// ---- Data types/METS/_StationOperational/C715 Tempalate Example/E_04_ElevatorState_C715.TcDUT
TYPE E_04_ElevatorState_C715 :
(
	SEQ_04_INIT									:=0,
	SEQ_04_ENABLEDEVICES							:=1,
	SEQ_04_HOMING								:=10,
	SEQ_04_MOVETODOWNLIMIT_DONE				:=20,
	SEQ_04_HOMINGWITHDATUM						:=30,

	SEQ_04_MOVETOHOMEPOS_TRY					:=40,
	SEQ_04_MOVETOHOMEPOS_DONE					:=50,
	SEQ_04_HOMED								:=90,
	SEQ_04_READY									:=100,

	SEQ_04_REQACCEPTED							:=110,

	SEQ_04_MOVEUP_TRY							:=120,
	SEQ_04_MOVEUP_DONE							:=130,
	SEQ_04_UNLOADBUNDLE_TRY						:=140,
	SEQ_04_UNLOADBUNDLE_DONE					:=150,

	SEQ_04_MOVEPOSITIVE_TRY						:=160,
	SEQ_04_MOVEPOSITIVE_DONE						:=170,
	SEQ_04_MOVENEGATIVE_TRY						:=180,
	SEQ_04_MOVENEGATIVE_DONE					:=190,
	SEQ_04_REJECTEXTEND_TRY						:=200,
	SEQ_04_REJECTEXTEND_DONE						:=210,
	SEQ_04_REJECTRETRACT_TRY						:=220,
	SEQ_04_REJECTRETRACT_DONE						:=230,


	(*SEQ_04_MOVEDOWN_TRY						:=160,
	SEQ_04_MOVEDOWN_DONE						:=170,*)

	SEQ_04_COMPLETE_TRY							:=340,
	SEQ_04_COMPLETE								:=350

);
END_TYPE

// ---- Data types/METS/_StationOperational/C715 Tempalate Example/E_Axis_C715.TcDUT
TYPE E_Axis_C715 :
(
	E_C715_WALKINGBEAM	:=1,
	E_C715_ELEVATOR		:=2,
	E_C715_TRANSFER		:=3,
	E_C715_PRESENTATION	:=4

);
END_TYPE

// ---- Data types/METS/_StationOperational/C715 Tempalate Example/E_Cylinder_C715.TcDUT
TYPE E_Cylinder_C715 :
(
	E_C715_STOPGATE01		:=1,
	E_C715_STOPGATE02		:=2,
	E_C715_BUNDLEALIGN	:=3,
	E_C715_TAMPHEAD		:=4,
	E_C715_LABELFORM		:=5,
	E_C715_BUNDLEREJECT	:=6,
	E_C715_BUNDLEPUSH	:=7

);
END_TYPE

// ---- Data types/METS/_StationOperational/C715 Tempalate Example/ST_04_ElevatorSeq_C715.TcDUT
  TYPE ST_04_ElevatorSeq_C715 :
STRUCT
	e04SeqState					: E_04_ElevatorState_C715;

	bSeqAbort					:BOOL;		(*Function Abort By Manager*)
	bSeqHomingRequest			:BOOL;		(*FUNCTION Homing Requested BY Manager OR Internal Functions*)
	bSeqWaitOnRequest			:BOOL;		(*Function In Valide State Avaiting For Request Command*)
	bSeqRequest					:BOOL;		(*Request Commnad To Start Function Cycle*)

	bSeqIsHoming					: BOOL;
	bSeqInProgress				:BOOL;		(*Function In Progress With Cycle*)
	bSeqComplete				:BOOL;		(*Function Complete Cycle - Flag Set After Every Cycle Finsh*)
	bSeqDone					:BOOL;		(*Function Sequence Finished With Success - Flag Set For One PLC Cycle*)
	bSeqError						: BOOL;
	nSeqErrorID					: UDINT;

	bAutoHomingAllowed			: BOOL;
	bStationHomed					:BOOL;		(*FUNCTION Homed*)
	bStationNotMoving				:BOOL;		(*Function Parts Are Not Moving*)
	bStationInPause				: BOOL;

	bMachineInError				: BOOL;
	bPassthroughMode				:BOOL;

	stBundleTracking				: ST_BundleTrackingRegister_C715;
	bTrackigDataSync				: BOOL;
	bDisableBottomLimit			: BOOL;

	bSynchroMoveActive			: BOOL;

END_STRUCT
END_TYPE

// ---- Data types/METS/_StationOperational/C715 Tempalate Example/ST_BundleTrackingRegister_C715.TcDUT
TYPE ST_BundleTrackingRegister_C715 :
STRUCT
	bOuterPresent				: BOOL;
	sOuterTimeStamp			: STRING(30);
	bOuterAligned				: BOOL;
	bLabelApplied				: BOOL;		(* TRUE = label has been printed and applied to Outer *)
	bLabelFormed				: BOOL;
	sLabelBarcode				: T_OUTER_Barcode;
	sConfirmationCode 			: T_MaxString;
	bOCVCreated				: BOOL;
	bOACCreated				: BOOL;
	bOuterIsValid				: BOOL;
	bDumpDataReq			: BOOL;
END_STRUCT
END_TYPE

// ---- Data types/METS/_StationOperational/C715 Tempalate Example/ST_CommonStationConfig_C715.TcDUT
TYPE ST_CommonStationConfig_C715 :
STRUCT

	fWalkingBeamHomeOffset		: LREAL :=55;
	fWalkingBeamVelo			: LREAL :=250;
	fWalkingBeamDistance		: LREAL :=360;

	tAlignTimeOut				: TIME  :=T#10S;

	tFormHeadTime				: TIME 	:=T#1500MS;

	fElevatorHomeOffset			: LREAL :=0;
	fElevatorMoveUpVelo			: LREAL :=400;
	fElevatorUnloadPosition		: LREAL :=310;
	fElevatorMoveDownVelo		: LREAL :=600;
	fElevatorLoadPosition		: LREAL :=0;

	tTransferTimeOut			: TIME 	:=T#10S;

	fTransferHomeOffset			: LREAL :=0;
	fTransferRejectVelo			: REAL 	:=-400;
	fTransferValidVelo			: REAL 	:=400;

	fPresentationHomeOffset		: LREAL :=0;
	fPresentationVelo			: REAL 	:=400;
	fPresentationDistance		: REAL 	:=115;

	(*bAllStationsHomed			: BOOL;
	bAllStationsCycledStopped	: BOOL;
	bCycleStopRequest			: BOOL;
	bManualModeHMI				: BOOL;
	bAllStationsOKToIndex		: BOOL;*)
END_STRUCT
END_TYPE

// ---- Data types/METS/_StationOperational/E_00_StationStateTemplate.TcDUT
TYPE E_00_StationStateTemplate :
(
	SEQ_00_INIT									:=0,
	SEQ_00_ENABLEDEVICES							:=1,
	SEQ_00_HOMING								:=10,
	SEQ_00_MOVETOHOMEPOS_TRY					:=20,
	SEQ_00_MOVETOHOMEPOS_DONE					:=30,
	SEQ_00_HOMED								:=90,
	SEQ_00_READY									:=100,

	SEQ_00_REQACCEPTED							:=110,

(***************************************************************************)
(**)
(***************************************************************************)

	SEQ_00_COMPLETE_TRY							:=340,
	SEQ_00_COMPLETE								:=350


);
END_TYPE

// ---- Data types/METS/_StationOperational/Manual Machine/E_OuterPrintStationState.TcDUT
TYPE E_OuterPrintStationState :
(
	STATION_SEQ_INIT:=100,
	STATION_SEQ_TRY_HOMING:=110,
	STATION_SEQ_HOMED:=120,
	STATION_SEQ_READY:=130,

	STATION_SEQ_GATE_DOWN_TRY:=140,
	STATION_SEQ_GATE_DOWN_DONE:=150,

	STATION_SEQ_APPLY_LABEL_TRY:=160,
	STATION_SEQ_APPLY_LABEL_DONE:=170,

	STATION_SEQ_GATE_UP_TRY:=180,
	STATION_SEQ_GATE_UP_DONE:=190,

	STATION_SEQ_COMPLETE_TRY:=200,
	STATION_SEQ_COMPLETE:=210


);
END_TYPE

// ---- Data types/METS/_StationOperational/SeqCtrl/ST_STATION_Requests.TcDUT
TYPE ST_STATION_Requests :
STRUCT

	bSeqAbort						:BOOL;		(*Function Abort By Manager*)
	bSeqInhibit						: BOOL;		(*in girafe is like bMachineInError*)
	bSeqHomingRequest			:BOOL;		(*FUNCTION Homing Requested BY Manager OR Internal Functions*)
	bSeqWaitOnRequest			:BOOL;		(*Function In Valide State Avaiting For Request Command*)
	bSeqRequest					:BOOL;		(*Request Commnad To Start Function Cycle*)

END_STRUCT
END_TYPE

// ---- Data types/METS/_StationOperational/SeqCtrl/ST_STATION_Status.TcDUT
TYPE ST_STATION_Status :
STRUCT

	bSeqIsHoming					: BOOL;
	bStationHomed					:BOOL;		(*FUNCTION Homed*)
	bSeqInProgress				:BOOL;		(*Function In Progress With Cycle*)
	bSeqComplete				:BOOL;		(*Function Complete Cycle - Flag Set After Every Cycle Finsh*)
	bSeqDone					:BOOL;		(*Function Sequence Finished With Success - Flag Set For One PLC Cycle*)
	bStationNotMoving				:BOOL;		(*Function Parts Are Not Moving*)

	bSeqError						: BOOL;
	nSeqErrorID					: UDINT;

END_STRUCT
END_TYPE

// ---- Data types/METS/_StationOperational/ST_00_StationStructTemplate.TcDUT
TYPE ST_00_StationStructTemplate :
STRUCT

	e00SeqState		: E_00_StationStateTemplate;

	REQ				: ST_STATION_Requests;
	STAT				: ST_STATION_Status;

(*Variable examles only*)
(*
	bPassthroughMode			:BOOL;

	stBundleTracking				: ST_BundleTrackingRegister;
	bTrigCamera					: BOOL;
	bCameraDone					: BOOL;


*)

END_STRUCT
END_TYPE

// ---- POUs/_Exclude/DUT/E_LOG_HandlerName_OLD.TcDUT
TYPE E_LOG_HandlerName_OLD :
(

		//E_LOG_OKCONECCTIONTOFSS,
		//E_LOG_LOSTCONECCTIONTOFSS,
		//E_LOG_DOOROPENZONE1,
		//E_LOG_DOOROPENZONE2,
		//E_LOG_STARTBUTTONPRESSED,
		//E_LOG_STOPBUTTONPRESSED,
		//E_LOG_RESETBUTTONPRESSED,
		//E_LOG_EUCANOTRUNNINGPT,
		//E_LOG_EUCANOTRUNNINGCT,
		//E_LOG_TPDNOTRUNNINGPT,
		//E_LOG_TPDNOTRUNNINGCT,
		//E_LOG_EXTNOTRUNNINGPT,
		//E_LOG_EXTNOTRUNNINGCT,
		//E_LOG_MACHINESTATEPT,
		//E_LOG_MACHINESTATECT,
		//E_LOG_PA1ADDED,
		//E_LOG_PA2ADDED,
		//E_LOG_PA3ADDED,
		//E_LOG_INTERIMDIAG1,
		//E_LOG_INTERIMDIAG2,
		//E_LOG_INTERIMDIAG3,
		//E_LOG_STACKOUTOFSEQ,
		//E_LOG_OUTERCOMPLETE,
		//E_LOG_LASTOCVCONTENT,
		//E_LOG_LASTPRINTER04COMMAND,
		//E_LOG_LASTPRINTER05COMMAND,
		//E_LOG_LASTOACCONTENT,
		//E_LOG_ROWCOMPLETE,
		//E_LOG_LAYERCOMPLETE,
		//E_LOG_INTERMEDIATECOMPLETE,
		//E_LOG_CASECOMPLETE,
		//E_LOG_CASEDISCHARGERT,
		//E_LOG_CASEDISCHARGEFT,
		//E_LOG_CASELABELVALIDATION,
		//E_LOG_OUTERAGGREGATIONCODE,
		//E_LOG_ROWCOMPLETECODES,
		//E_LOG_LAYERCOMPLETECODES,
		//E_LOG_FINALISECASECONTENTCODES,
		//E_LOG_INTERPUSHOVERWIRTTEN,
		//E_LOG_CASECOMPLETEOVERWITTEN,
		//E_LOG_CASEDISCHARGEOVERWRITTEN,
		//E_LOG_REJECTEDBYCASEPACKER,
		//E_LOG_CASELABELCODE,
		//E_LOG_MCCREATEDEVENT,
		//E_LOG_CASEVALIDATIONRT,
		//E_LOG_CASEVALIDATIONFT,
		//E_LOG_OCVWRITEERROR,
		//E_LOG_OACWRITEERROR,
		//E_LOG_CACWRITEERROR,
		//E_LOG_CHMWRITEERROR,
		//E_LOG_MLFILLINSTATUS,
		//E_LOG_MLSTATUS,
		//E_LOG_MLRESOTRESTATUS,
		//E_LOG_CODEDIAG1,
		//E_LOG_CODEDIAG2,
		//E_LOG_CODEDIAG3,
		//E_LOG_CODEDIAG4,
		//E_LOG_MASTERLISTDOOR,
		//E_LOG_AGGREGATIONDOOR,
		//E_LOG_WRAPPERDOOR,
		//E_LOG_WRAPPERREJECT1
		//E_LOG_WRAPPERREJECT2



);
END_TYPE

// ---- POUs/_Exclude/DUT/ST_SYSTEM_Config_old.TcDUT
TYPE ST_SYSTEM_Config_old :
STRUCT
(*General EUCA-TPD*)
	sBackupName								: STRING;
	sProductionSite 							: STRING(4);
	stProductionLine 							: ST_SYSTEM_ProductionLine;
	sShiftOffsetTime							: STRING(6);	(* shift offset time, formatted as '-06:00' or '+02:00' *)
	stSoftVersion								: ST_SYSTEM_SoftwareVersion;
	bEUCAMonitor24VSupply					: BOOL := TRUE;
	bMonitorRemote24VSupply				: BOOL;
	bInhibitSafetyResetWhenAirNOK			: BOOL;

	bConditionalStateAllowed					: BOOL := TRUE;
	bNoStationsAvailable						: BOOL := TRUE;

	nPackAggregationMode						: INT :=0; (* 0 -NOPACKAGGREGATION, 1 -STRUCTURALAGGREGATION (PAOL), 2 -STRUCTURALAGGREGATION (2CAM),  3 - LINEARAGGREGATION (PLAS), 4 - NCWAGGREGATION (PLAS + INTERIM)*)
	nOuterAggregationMode						: INT := 0; (* 0 - SYNCHROCONFIRMATION, 1 - SHIFTCONFIRMATION, 2 -SFLXNOCONFIRMATION, 3 - SFLXWITHCONFIRMATION, 4 - LASERPRINTLABEL*)
	nAutomationMode								: INT := 0; (* 0 - EXTERNAL, 1 - CML, 2 - LARS, 3 - SIDEFLEX *)

(*FSS settings*)
	tFSSLostConnectionTimeOut				: TIME := t#30m;
	sFSS_Server_IPAddress						: STRING:= '127.0.0.1'; (*Do not remove. Used for HMI*)
	sFSS_Server_WebRequest					: T_MaxString := 'http://127.0.0.1/Apriso/MessageProcessor/FlexNetMessageProcessor.asmx'; (*Do not removed. Used for HMI - this is the CHM sending endpoint*)
	nFSSResponseTimeout						: UINT := 60000; (*: TIME := t#60s;*)
	nFSSResendAttempts						: INT := 5;

	bKPIRemoteShareEnable					: BOOL;
	bSystemLogEnable							: BOOL := TRUE;
	bExtendedDiagnosticEnable				: BOOL;

	bPAOLIsolatorExist						: BOOL;
	bLightbox4TrigerSystemExist				: BOOL;
	bLightboxLensAirExist						: BOOL;
	tLightboxLensAirFrequency				: TIME:=t#3h;
	tLightboxLensAirBlowDuration			: TIME:=t#10s;

	bLighboxOverCMLConveyor					: BOOL;
	bLightboxCamerasOnFullResolution				: BOOL;

	nAggregationUnitLightingIntensityTop				: INT := 100;		(*to be removed and replaced with camera config*)
	nAggregationUnitLightingIntensity			: INT := 100;				(*to be removed and replaced with camera config*)
	(*nConfirmationUnitLightingIntensity			: INT := 100;				(*to be removed and replaced with camera config*)
	nMasterListLightingIntensity				: INT := 100;	*)				(*to be removed and replaced with camera config*)

	bExistWrapperPackRejectSesnor					: BOOL;
	bFrontConfirmationCameraInUse			: BOOL;				(*Rear confirmation camera 192.168.1.41 = false, front confiramtion camera 192.168.1.42 = true*)

	sFC1ReplacmentChar						: STRING(1) := '';
	bATTPModeEnable							: BOOL := TRUE;

	bCloseCameraRelay						: BOOL;
	bPassthrough								: BOOL;
	bPassthroughTPD							: BOOL;
	tPassthroughDisableDelay					: TIME := t#2000ms;
	bApplyLabelInPassthrough					: BOOL;
	bDisableApplyLabel						: BOOL;
	bPrinterHighSpeedEnable					: BOOL;
	bEANValidationEnable						: BOOL;
	bValidateOCVOnly							: BOOL;
	bPrintSignalFromPLC						: BOOL;
	bEnableResendCommand					: BOOL;


(*Camera - IP/Port settings for All scanners used in EUCA-TPD  arrays with up to 6 scanners per array *)
	aCameraSettings							: ARRAY[1..cMAX_CAMERA_NUMBER] OF ST_SCANNER_Config;

(*Printers*)
	aPrinterSettings							: ARRAY[1..cMAX_PRINTER_NUMBER] OF ST_PRINTER_Config;

(*Hand Scanners*)
	aHandScannersConfig						: ARRAY[1..cMAX_HAND_SCANNERS] OF ST_SCANNER_HoneywellConfig;
	aHoneywellCtrl								: ARRAY[1..cMAX_HAND_SCANNERS] OF ST_SCANNER_HoneywellCtrl;
	stUSBScannerConfig						: ST_SCANNER_USBConfig;
	bHandScannerInMainCabinet				: BOOL; (*to be tested*)

(* Profinet drives *)
	aProfiNetMaster							: ARRAY [1..cMAX_PROFINET_MASTERS]  OF  ST_ProfinetMasterConfig; (* EL6631 *)
	aProfiNetDrive								: ARRAY [1..cMAX_PROFINET_DRIVES]  OF ST_ProfinetDrive; (*config for individual drives *)

(*MC2 drives*)
	aAxisConfig								: ARRAY[1..cMAX_MC2_DRIVES] OF ST_AXIS_Config;

(* Analog drive*)
	bPackSeparatorAnalogControl				: BOOL;
	stPackSeparator							: ST_AnalogDrive;

(* CAMS  *)
	(*aAFS50camConfig							: ARRAY [1.. cMAX_CAMS] OF ST_AFS60_Config;*)

(*Cylinders*)
	aCylinderConfig							: ARRAY[1..cMAX_CYLINDERS] OF ST_CYLINDER_Config;

(* Consecutive rejects counter*)
	nConsecutivePackRejects						: UINT := 3;
	nConsecutivePackConfirmationMissing			: UINT := 3;
	nConsecutiveOCVMissing						: UINT := 3;
	nConsecutiveIntermediateNoRead				: UINT := 3;
	nConsecutiveOuterRejects					: UINT := 3;
	nConsecutiveCaseContentMissing				: UINT := 3;
	nConsecutiveCaseRejects						: UINT := 3;

(*Barcode setup - NEW - Gradually implementing*)
	stCodeInfo_Pack								: ST_CodeInfo :=		(eCodeType :=E_PACK);
	stCodeInfo_Intermediate						: ST_CodeInfo :=		(eCodeType :=E_INTERIM);
	stCodeInfo_Outer								: ST_CodeInfo :=		(eCodeType :=E_OUTER);
	stCodeInfo_Case								: ST_CodeInfo :=		(eCodeType :=E_CASE);

(*bExistInfeedConveyorStartSensor			:BOOL;*)
	bExistPreTPDBuildBackSensor					: BOOL := TRUE;
	bExistTPDExitBlockedSensor					: BOOL := TRUE;
	bExistPreEUCABuildBackSensor				: BOOL;
	bExistEUCAExitBlockedSensor					: BOOL;

	bConveyorAsPreMachine						: BOOL := TRUE;

(*Enable Restoring of OCV data from structure*)
	bEnableRestoreOCV							: BOOL;

(*Enable arming sensors even if outer did not leave Lightox yet *)
	bEnableFastArming							: BOOL:=TRUE;

(*Enable Master List Fillin*)
	bEnablePackPrimaryMasterList					: BOOL:=TRUE;
	bEnablePackSecondaryMasterList				: BOOL:=TRUE;
	bEnableOuterMasterList						: BOOL:=TRUE;

	nClearPMLIndex								: INT;
	nClearPMLRecords								: INT;

(*Commisioning settings*)
	bEnableOuterRejectConfirmation			: BOOL;
	bEnableOuterTransferConfirmation		: BOOL;
	bDisableOuterReject						: BOOL;	(*Disable any outer reject - just for commisioning*)
	bDisableCaseReject						: BOOL;	(*Disable any case reject - just for commisioning*)
	bOuterRejectWithHighSignal				: BOOL;
	bCaseRejectWithHighSignal				: BOOL;
	bCommisioningMode						: BOOL; 	(*Write CHM file but  don't send to FSS, use by HMI, do not delete*)

(*Database*)
	(*stDBConfig								: ST_DB_Config;*)

(*Door*)
	stDoorSettingsZone1					: ST_SYSTEM_Door;
	stDoorSettingsZone2					: ST_SYSTEM_Door;

(*******************************************************************************************************************************************************)
(*Single Input Config*)
	st_I_TransferCoveyorDoorGuard1			: ST_IO2_SingleInputCtrl:=			(eTypeInput:=NO,		tTimeOnFilter:=t#100ms, 		tTimeOffFilter:=t#10ms, 	sInputName:='Transfer Coveyor Door Guard 1' );	(**)
	st_I_TransferCoveyorDoorGuard2			: ST_IO2_SingleInputCtrl:=			(eTypeInput:=NO,		tTimeOnFilter:=t#100ms, 		tTimeOffFilter:=t#10ms, 	sInputName:='Transfer Coveyor Door Guard 2' );	(**)

	st_I_DoorOpenZone1					: ST_IO2_SingleInputCtrl:=			(eTypeInput:=NO,		tTimeOnFilter:=t#100ms, 		tTimeOffFilter:=t#10ms, 	sInputName:='Door Open Zone 1' );	(**)
	st_I_DoorOpenZone2					: ST_IO2_SingleInputCtrl:=			(eTypeInput:=NO,		tTimeOnFilter:=t#100ms, 		tTimeOffFilter:=t#10ms, 	sInputName:='Door Open Zone 2' );	(**)

	st_I_AuxRowCompleteSesnor			: ST_IO2_SingleInputCtrl:=			(eTypeInput:=NO,		tTimeOnFilter:=t#10ms, 		tTimeOffFilter:=t#10ms, 	sInputName:='Aux Row Complete' );	(**)
	st_I_CaseRejectedByCasePacker		: ST_IO2_SingleInputCtrl:=			(eTypeInput:=NO,		tTimeOnFilter:=t#10ms, 		tTimeOffFilter:=t#10ms, 	sInputName:='Case Rejected By Casepacker' );	(**)

	st_I_PreMachineAutoRun				: ST_IO2_SingleInputCtrl:=			(eTypeInput:=NO,		tTimeOnFilter:=t#100ms, 		tTimeOffFilter:=t#0ms, 	sInputName:='PreMachine AutoRun' );	(**)
	st_I_CasePackerAutoRun				: ST_IO2_SingleInputCtrl:=			(eTypeInput:=NO,		tTimeOnFilter:=t#100ms, 		tTimeOffFilter:=t#0ms, 	sInputName:='Casepacker AutoRun' );	(**)

	st_I_QAButtonRejectOuter				: ST_IO2_SingleInputCtrl:=			(eTypeInput:=NO,		tTimeOnFilter:=t#100ms, 		tTimeOffFilter:=t#0ms, 	sInputName:='QA Button Reject Outer' );	(**)
	st_I_OuterAtRejectStation				: ST_IO2_SingleInputCtrl:=			(eTypeInput:=NO,		tTimeOnFilter:=t#1000ms, 		tTimeOffFilter:=t#0ms, 	sInputName:='Outer At Reject Station' );	(**)
	st_I_OuterRejectConfirm				: ST_IO2_SingleInputCtrl:=			(eTypeInput:=NO,		tTimeOnFilter:=t#1000ms, 		tTimeOffFilter:=t#0ms, 	sInputName:='Outer Reject Confirm' );	(**)
	st_I_RejectBinFull					: ST_IO2_SingleInputCtrl:=			(eTypeInput:=NO,		tTimeOnFilter:=t#100ms, 		tTimeOffFilter:=t#0ms, 	sInputName:='Reject Bin Full' );	(**)

	st_I_EUCABuildBackPreMachine			: ST_IO2_SingleInputCtrl:=			(eTypeInput:=NO,		tTimeOnFilter:=t#1000ms, 		tTimeOffFilter:=t#0ms, 	sInputName:='EUCA Buildback Sensor' );	(**)
	st_I_EUCAExitBlocked					: ST_IO2_SingleInputCtrl:=			(eTypeInput:=NO,		tTimeOnFilter:=t#1000ms, 		tTimeOffFilter:=t#0ms, 	sInputName:='EUCA Exit Blocked Sensor' );	(**)

	st_I_OuterAtSystemInfeed				: ST_IO2_SingleInputCtrl:=			(eTypeInput:=NO,		tTimeOnFilter:=t#1000ms, 		tTimeOffFilter:=t#0ms, 	sInputName:='Outer At System Infeed Sensor' );	(**)
	st_I_OuterAtAdditionalConv				: ST_IO2_SingleInputCtrl:=			(eTypeInput:=NO,		tTimeOnFilter:=t#1000ms, 		tTimeOffFilter:=t#0ms, 	sInputName:='Outer At Additional Conv Sensor' );	(**)

	st_I_TransferConveyorPlugConnected		: ST_IO2_SingleInputCtrl:=			(eTypeInput:=NO,		tTimeOnFilter:=t#100ms, 		tTimeOffFilter:=t#100ms, 	sInputName:='Transfer Conveyor Plug Connected' );	(**)
	st_I_OutfeedConveyorPlugConnected		: ST_IO2_SingleInputCtrl:=			(eTypeInput:=NO,		tTimeOnFilter:=t#100ms, 		tTimeOffFilter:=t#100ms, 	sInputName:='Outfeed Conveyor Plug Connected' );	(**)
	st_I_AdditionalConveyorPlugConnected	: ST_IO2_SingleInputCtrl:=			(eTypeInput:=NO,		tTimeOnFilter:=t#100ms, 		tTimeOffFilter:=t#100ms, 	sInputName:='Outfeed Conveyor Plug Connected' );	(**)

(*Single Input Config for camera triggers*)

	st_I_Camera01						: ST_IO2_SingleInputCtrl:=			(eTypeInput:=NO,		tTimeOnFilter:=t#6ms, 		tTimeOffFilter:=t#20ms, 	sInputName:='Camera 01' );	(**)
	st_I_Camera02						: ST_IO2_SingleInputCtrl:=			(eTypeInput:=NO,		tTimeOnFilter:=t#6ms, 		tTimeOffFilter:=t#20ms, 	sInputName:='Camera 02' );	(**)
	st_I_Camera03						: ST_IO2_SingleInputCtrl:=			(eTypeInput:=NO,		tTimeOnFilter:=t#6ms, 		tTimeOffFilter:=t#20ms, 	sInputName:='Camera 03' );	(**)
	st_I_Camera04						: ST_IO2_SingleInputCtrl:=			(eTypeInput:=NO,		tTimeOnFilter:=t#10ms, 		tTimeOffFilter:=t#0ms, 	sInputName:='Camera 04' );	(**)
	st_I_Camera05						: ST_IO2_SingleInputCtrl:=			(eTypeInput:=NO,		tTimeOnFilter:=t#10ms, 		tTimeOffFilter:=t#0ms, 	sInputName:='Camera 05' );	(**)
	st_I_Camera06						: ST_IO2_SingleInputCtrl:=			(eTypeInput:=NO,		tTimeOnFilter:=t#10ms, 		tTimeOffFilter:=t#0ms, 	sInputName:='Camera 06' );	(**)
	st_I_Camera07						: ST_IO2_SingleInputCtrl:=			(eTypeInput:=NO,		tTimeOnFilter:=t#10ms, 		tTimeOffFilter:=t#0ms, 	sInputName:='Camera 07' );	(**)
	st_I_Camera08						: ST_IO2_SingleInputCtrl:=			(eTypeInput:=NO,		tTimeOnFilter:=t#10ms, 		tTimeOffFilter:=t#0ms, 	sInputName:='Camera 08' );	(**)
	st_I_Camera09						: ST_IO2_SingleInputCtrl:=			(eTypeInput:=NO,		tTimeOnFilter:=t#10ms, 		tTimeOffFilter:=t#0ms, 	sInputName:='Camera 09' );	(**)
	st_I_Camera10						: ST_IO2_SingleInputCtrl:=			(eTypeInput:=NO,		tTimeOnFilter:=t#10ms, 		tTimeOffFilter:=t#0ms, 	sInputName:='Camera 10' );	(**)
	st_I_Camera11						: ST_IO2_SingleInputCtrl:=			(eTypeInput:=NO,		tTimeOnFilter:=t#10ms, 		tTimeOffFilter:=t#0ms, 	sInputName:='Camera 11' );	(**)
	st_I_Camera12						: ST_IO2_SingleInputCtrl:=			(eTypeInput:=NO,		tTimeOnFilter:=t#10ms, 		tTimeOffFilter:=t#0ms, 	sInputName:='Camera 12' );	(**)

(*METS Cylinders Filtered Inputs *)

	st_I_ClampCylinderExtended		: ST_IO2_SingleInputCtrl:=			(eTypeInput:=NO,		tTimeOnFilter:=t#10ms, 		tTimeOffFilter:=t#0ms, 	sInputName:='Clamp Cylinder Extended' );	(**)
	st_I_ClampCylinderRetracted		: ST_IO2_SingleInputCtrl:=			(eTypeInput:=NO,		tTimeOnFilter:=t#10ms, 		tTimeOffFilter:=t#0ms, 	sInputName:='Clamp Cylinder Retracted' );	(**)

	st_I_GateCylinderExtended		: ST_IO2_SingleInputCtrl:=			(eTypeInput:=NO,		tTimeOnFilter:=t#10ms, 		tTimeOffFilter:=t#0ms, 	sInputName:='Gate Cylinder Extended' );	(**)
	st_I_GateCylinderRetracted 		: ST_IO2_SingleInputCtrl:=			(eTypeInput:=NO,		tTimeOnFilter:=t#10ms, 		tTimeOffFilter:=t#0ms, 	sInputName:='Gate Cylinder Retracted' );	(**)

	st_I_RejectCylinderExtended		: ST_IO2_SingleInputCtrl:=			(eTypeInput:=NO,		tTimeOnFilter:=t#10ms, 		tTimeOffFilter:=t#0ms, 	sInputName:='Reject Cylinder Extended' );	(**)
	st_I_RejectCylinderRetracted 		: ST_IO2_SingleInputCtrl:=			(eTypeInput:=NO,		tTimeOnFilter:=t#10ms, 		tTimeOffFilter:=t#0ms, 	sInputName:='Reject Cylinder Retracted' );	(**)

	st_I_AdditionalRejectCylinderExtended		: ST_IO2_SingleInputCtrl:=			(eTypeInput:=NO,		tTimeOnFilter:=t#10ms, 		tTimeOffFilter:=t#0ms, 	sInputName:='Reject Cylinder Extended' );	(**)
	st_I_AdditionalRejectCylinderRetracted 		: ST_IO2_SingleInputCtrl:=			(eTypeInput:=NO,		tTimeOnFilter:=t#10ms, 		tTimeOffFilter:=t#0ms, 	sInputName:='Reject Cylinder Retracted' );	(**)

	st_I_FirstPusherCylinderExtended		: ST_IO2_SingleInputCtrl:=			(eTypeInput:=NO,		tTimeOnFilter:=t#10ms, 		tTimeOffFilter:=t#0ms, 	sInputName:='Reject Cylinder Extended' );	(**)
	st_I_FirstPusherCylinderRetracted 		: ST_IO2_SingleInputCtrl:=			(eTypeInput:=NO,		tTimeOnFilter:=t#10ms, 		tTimeOffFilter:=t#0ms, 	sInputName:='Reject Cylinder Retracted' );	(**)

	st_I_SecondPusherCylinderExtended		: ST_IO2_SingleInputCtrl:=			(eTypeInput:=NO,		tTimeOnFilter:=t#10ms, 		tTimeOffFilter:=t#0ms, 	sInputName:='Reject Cylinder Extended' );	(**)
	st_I_SecondPusherCylinderRetracted 		: ST_IO2_SingleInputCtrl:=			(eTypeInput:=NO,		tTimeOnFilter:=t#10ms, 		tTimeOffFilter:=t#0ms, 	sInputName:='Reject Cylinder Retracted' );	(**)

(*METS Labellers Filtered Inputs *)

	st_I_Labeller1InPosition					: ST_IO2_SingleInputCtrl:=			(eTypeInput:=NO,		tTimeOnFilter:=t#10ms, 		tTimeOffFilter:=t#0ms, 	sInputName:='Labeller1 In Position' );	(**)
	st_I_Labeller1OuterAtLabeller				: ST_IO2_SingleInputCtrl:=			(eTypeInput:=NO,		tTimeOnFilter:=t#10ms, 		tTimeOffFilter:=t#0ms, 	sInputName:='Labeller1 Outer At Labeller' );	(**)
	tLabeller1OuterAtLabellerTimeLatch		: TIME := t#200ms; (*Variable used separately to keep one standard with HMI user controls for Single Inputs*)

	st_I_Labeller1Ready						: ST_IO2_SingleInputCtrl:=			(eTypeInput:=NO,		tTimeOnFilter:=t#10ms, 		tTimeOffFilter:=t#0ms, 	sInputName:='Labeller1 Ready' );	(**)
	st_I_Labeller1DataReady					: ST_IO2_SingleInputCtrl:=			(eTypeInput:=NO,		tTimeOnFilter:=t#10ms, 		tTimeOffFilter:=t#0ms, 	sInputName:='Labeller1 Data Ready' );	(**)
	st_I_Labeller1HomePosition				: ST_IO2_SingleInputCtrl:=			(eTypeInput:=NO,		tTimeOnFilter:=t#10ms, 		tTimeOffFilter:=t#0ms, 	sInputName:='Labeller1 Home Position' );	(**)
	st_I_Labeller1LabelPrinted					: ST_IO2_SingleInputCtrl:=			(eTypeInput:=NO,		tTimeOnFilter:=t#10ms, 		tTimeOffFilter:=t#0ms, 	sInputName:='Labeller1 Label Printed' );	(**)
	st_I_Labeller1ReadyToApply				: ST_IO2_SingleInputCtrl:=			(eTypeInput:=NO,		tTimeOnFilter:=t#10ms, 		tTimeOffFilter:=t#0ms, 	sInputName:='Labeller1 Ready To Apply' );	(**)
	st_I_Labeller1ApplyDone					: ST_IO2_SingleInputCtrl:=			(eTypeInput:=NO,		tTimeOnFilter:=t#10ms, 		tTimeOffFilter:=t#0ms, 	sInputName:='Labeller1 Apply Done' );	(**)
	st_I_Labeller1SummaryWarning			: ST_IO2_SingleInputCtrl:=			(eTypeInput:=NO,		tTimeOnFilter:=t#10ms, 		tTimeOffFilter:=t#0ms, 	sInputName:='Labeller1 Summary Warning' );	(**)
	st_I_Labeller1Error							: ST_IO2_SingleInputCtrl:=			(eTypeInput:=NO,		tTimeOnFilter:=t#10ms, 		tTimeOffFilter:=t#0ms, 	sInputName:='Labeller1 Error' );	(**)


	st_I_Labeller2InPosition					: ST_IO2_SingleInputCtrl:=			(eTypeInput:=NO,		tTimeOnFilter:=t#10ms, 		tTimeOffFilter:=t#0ms, 	sInputName:='Labeller2 In Position' );	(**)
	st_I_Labeller2OuterAtLabeller				: ST_IO2_SingleInputCtrl:=			(eTypeInput:=NO,		tTimeOnFilter:=t#10ms, 		tTimeOffFilter:=t#0ms, 	sInputName:='Labeller2 Outer At Labeller' );	(**)
	tLabeller2OuterAtLabellerTimeLatch		: TIME := t#40ms; (*Variable used separately to keep one standard with HMI user controls for Single Inputs*)

	st_I_Labeller2Ready						: ST_IO2_SingleInputCtrl:=			(eTypeInput:=NO,		tTimeOnFilter:=t#10ms, 		tTimeOffFilter:=t#0ms, 	sInputName:='Labeller2 Ready' );	(**)
	st_I_Labeller2DataReady					: ST_IO2_SingleInputCtrl:=			(eTypeInput:=NO,		tTimeOnFilter:=t#10ms, 		tTimeOffFilter:=t#0ms, 	sInputName:='Labeller2 Data Ready' );	(**)
	st_I_Labeller2HomePosition				: ST_IO2_SingleInputCtrl:=			(eTypeInput:=NO,		tTimeOnFilter:=t#10ms, 		tTimeOffFilter:=t#0ms, 	sInputName:='Labeller2 Home Position' );	(**)
	st_I_Labeller2LabelPrinted					: ST_IO2_SingleInputCtrl:=			(eTypeInput:=NO,		tTimeOnFilter:=t#10ms, 		tTimeOffFilter:=t#0ms, 	sInputName:='Labeller2 Label Printed' );	(**)
	st_I_Labeller2ReadyToApply				: ST_IO2_SingleInputCtrl:=			(eTypeInput:=NO,		tTimeOnFilter:=t#10ms, 		tTimeOffFilter:=t#0ms, 	sInputName:='Labeller2 Ready To Apply' );	(**)
	st_I_Labeller2ApplyDone					: ST_IO2_SingleInputCtrl:=			(eTypeInput:=NO,		tTimeOnFilter:=t#10ms, 		tTimeOffFilter:=t#0ms, 	sInputName:='Labeller2 Apply Done' );	(**)
	st_I_Labeller2SummaryWarning			: ST_IO2_SingleInputCtrl:=			(eTypeInput:=NO,		tTimeOnFilter:=t#10ms, 		tTimeOffFilter:=t#0ms, 	sInputName:='Labeller2 Summar yWarning' );	(**)
	st_I_Labeller2Error							: ST_IO2_SingleInputCtrl:=			(eTypeInput:=NO,		tTimeOnFilter:=t#10ms, 		tTimeOffFilter:=t#0ms, 	sInputName:='Labeller2 Error' );	(**)

(*METS SADDLE (Gating&Reject System) Filtered Inputs  FB***************************************************************************************************************)

	st_I_OuterAtClamp					: ST_IO2_SingleInputCtrl:=			(eTypeInput:=NO,		tTimeOnFilter:=t#100ms, 		tTimeOffFilter:=t#100ms, 		sInputName:='Outer At Clamp');	(**)
	st_I_OuterAtLabelGate				: ST_IO2_SingleInputCtrl:=			(eTypeInput:=NO,		tTimeOnFilter:=t#100ms, 		tTimeOffFilter:=t#100ms, 		sInputName:='Outer At Label Gate');	(**)
	st_I_GateClear						: ST_IO2_SingleInputCtrl:=			(eTypeInput:=NO,		tTimeOnFilter:=t#100ms, 		tTimeOffFilter:=t#100ms, 		sInputName:='Gate Clear');	(**)
	st_I_GateImpact					: ST_IO2_SingleInputCtrl:=			(eTypeInput:=NO,		tTimeOnFilter:=t#100ms, 		tTimeOffFilter:=t#100ms, 		sInputName:='Gate Impact');	(**)

(* Single Inputs for METS CML*)

	st_I_RotaryTransferPackAtStopPlate		: ST_IO2_SingleInputCtrl:=			(eTypeInput:=NO,		tTimeOnFilter:=t#1000ms, 		tTimeOffFilter:=t#0ms, 	sInputName:='Rotary Transfer Outer At Stop Plate');	(**)
	st_I_RotaryTransferTorqueLimiter			: ST_IO2_SingleInputCtrl:=			(eTypeInput:=NO,		tTimeOnFilter:=t#1000ms, 		tTimeOffFilter:=t#0ms, 	sInputName:='Rotary Transfer Torque Limiter');	(**)
	st_I_RotaryTransferDelayStop1			: ST_IO2_SingleInputCtrl:=			(eTypeInput:=NO,		tTimeOnFilter:=t#1000ms, 		tTimeOffFilter:=t#0ms, 	sInputName:='Rotary Transfer Delay Stop1');	(**)
	st_I_RotaryTransferDelayStop2			: ST_IO2_SingleInputCtrl:=			(eTypeInput:=NO,		tTimeOnFilter:=t#1000ms, 		tTimeOffFilter:=t#0ms, 	sInputName:='Rotary Transfer Delay Stop2');	(**)
	st_I_ConveyorIndexContact				: ST_IO2_SingleInputCtrl:=			(eTypeInput:=NO,		tTimeOnFilter:=t#50ms, 		tTimeOffFilter:=t#50s, 	sInputName:='Infeed Conveyor Start');	(**)
	st_I_Guard4ElectricalBoxInPosition		: ST_IO2_SingleInputCtrl:=			(eTypeInput:=NC,		tTimeOnFilter:=t#50ms, 		tTimeOffFilter:=t#50s, 	sInputName:='Electrical Box In Position Sensor');	(**)

(* Single Inputs for METS Manual Machine*)

	st_I_InfeedConveyorStart				: ST_IO2_SingleInputCtrl:=			(eTypeInput:=NO,		tTimeOnFilter:=t#1000ms, 		tTimeOffFilter:=t#0ms, 	sInputName:='Infeed Conveyor Start');	(**)
	st_I_RejectChuteExitBlocked			: ST_IO2_SingleInputCtrl:=			(eTypeInput:=NO,		tTimeOnFilter:=t#1000ms, 		tTimeOffFilter:=t#0ms, 	sInputName:='Reject Chute Blocked');	(**)

(* Single Inputs for METS SFLX Machine*)

	st_I_OuterInfeedJam				: ST_IO2_SingleInputCtrl:=			(eTypeInput:=NO,		tTimeOnFilter:=t#1000ms, 		tTimeOffFilter:=t#0ms, 	sInputName:='Outer Infeed Jam' );	(**)
	(*st_I_PackAggregationCameraTrigger		: ST_IO2_SingleInputCtrl:=			(eTypeInput:=NO,		tTimeOnFilter:=t#1000ms, 		tTimeOffFilter:=t#0ms, 	sInputName:='Pack Aggregation Camera Trigger');*)	(**)
	st_I_OutfeedConveyorStart				: ST_IO2_SingleInputCtrl:=			(eTypeInput:=NO,		tTimeOnFilter:=t#1000ms, 		tTimeOffFilter:=t#0ms, 	sInputName:='Outfeed Conveyor Start');	(**)
	st_I_RejectConfirmationNCW				: ST_IO2_SingleInputCtrl:=			(eTypeInput:=NO,		tTimeOnFilter:=t#1000ms, 		tTimeOffFilter:=t#0ms, 	sInputName:='Reject Confirmation NCW');	(**)
	st_I_RejectBinFullNCW					: ST_IO2_SingleInputCtrl:=			(eTypeInput:=NO,		tTimeOnFilter:=t#1000ms, 		tTimeOffFilter:=t#0ms, 	sInputName:='Reject Bin Full NCW');	(**)
	st_I_OuterAtTransferReject			: ST_IO2_SingleInputCtrl:=			(eTypeInput:=NO,		tTimeOnFilter:=t#1000ms, 		tTimeOffFilter:=t#0ms, 	sInputName:='Outer At Transfer Reject');	(**)
	st_I_OuterAtSideFlexExit				: ST_IO2_SingleInputCtrl:=			(eTypeInput:=NO,		tTimeOnFilter:=t#1000ms, 		tTimeOffFilter:=t#0ms, 	sInputName:='Outer At Side Flex Exit');	(**)
	st_I_OuterAtPostMachineInfeed		: ST_IO2_SingleInputCtrl:=			(eTypeInput:=NO,		tTimeOnFilter:=t#1000ms, 		tTimeOffFilter:=t#0ms, 	sInputName:='Outer At PostMachine Infeed');	(**)

	st_I_Guard1FlexInfeedDoor				: ST_IO2_SingleInputCtrl:=			(eTypeInput:=NC,		tTimeOnFilter:=t#1000ms, 		tTimeOffFilter:=t#0ms, 	sInputName:='Guard 1 Flex Infeed Door');	(**)
	st_I_Guard3FlexRHDoor					: ST_IO2_SingleInputCtrl:=			(eTypeInput:=NO,		tTimeOnFilter:=t#200ms, 		tTimeOffFilter:=t#200ms, 	sInputName:='Guard 3 Flex RH Door');	(**)
	st_I_Guard4FlexPrinterDoor					: ST_IO2_SingleInputCtrl:=			(eTypeInput:=NO,		tTimeOnFilter:=t#200ms, 		tTimeOffFilter:=t#200ms, 	sInputName:='Guard 4 Flex Printer Door');	(**)
	st_I_Guard5FlexLHDoor					: ST_IO2_SingleInputCtrl:=			(eTypeInput:=NO,		tTimeOnFilter:=t#200ms, 		tTimeOffFilter:=t#200ms, 	sInputName:='Guard 5 Flex LH Door	');	(**)

(*Single Input for PACAN*)

(*	st_I_StackerArmAtBackwardPosition	: ST_IO2_SingleInputCtrl:=			(eTypeInput:=NO,		tTimeOnFilter:=t#10ms, 		tTimeOffFilter:=t#0ms, 	sInputName:='Stacker Arm At Backward Position');	(**)
	st_I_StackerArmInTopPosition			: ST_IO2_SingleInputCtrl:=			(eTypeInput:=NO,		tTimeOnFilter:=t#10ms, 		tTimeOffFilter:=t#0ms, 	sInputName:='Stacker Arm In Top Position');	(**)
	st_I_StackPresentSensor1				: ST_IO2_SingleInputCtrl:=			(eTypeInput:=NO,		tTimeOnFilter:=t#10ms, 		tTimeOffFilter:=t#0ms, 	sInputName:='Stack Present Sensor1');	(**)
	st_I_StackPresentSensor2				: ST_IO2_SingleInputCtrl:=			(eTypeInput:=NO,		tTimeOnFilter:=t#10ms, 		tTimeOffFilter:=t#0ms, 	sInputName:='Stack Present Sensor2');	(**)
	st_I_StackerTransferPusher			: ST_IO2_SingleInputCtrl:=			(eTypeInput:=NO,		tTimeOnFilter:=t#10ms, 		tTimeOffFilter:=t#0ms, 	sInputName:='Stacker Transfer Pusher');	(**)
	st_I_StackerTransferComplete			: ST_IO2_SingleInputCtrl:=			(eTypeInput:=NO,		tTimeOnFilter:=t#10ms, 		tTimeOffFilter:=t#0ms, 	sInputName:='Stacker Transfer Complete');	(**)
	st_I_OuterAtPACANRejectStation		: ST_IO2_SingleInputCtrl:=			(eTypeInput:=NO,		tTimeOnFilter:=t#100ms, 		tTimeOffFilter:=t#100ms, 	sInputName:='Outer At PACAN Reject Station');	(**)
*)
(*Single Input for PAOL*)

	st_I_TPDExitBlockedSensor			: ST_IO2_SingleInputCtrl:=			(eTypeInput:=NO,		tTimeOnFilter:=t#100ms, 		tTimeOffFilter:=t#0ms, 	sInputName:='PAOL Exit Blocked Sensor');	(**)
	st_I_PreMachineBuildBackSensor		: ST_IO2_SingleInputCtrl:=			(eTypeInput:=NO,		tTimeOnFilter:=t#100ms, 		tTimeOffFilter:=t#0ms, 	sInputName:='PAOL Buildback Sensor');	(**)
	st_I_PackAggregCameraRigSensor		: ST_IO2_SingleInputCtrl:=			(eTypeInput:=NO,		tTimeOnFilter:=t#6ms, 		tTimeOffFilter:=t#6ms, 	sInputName:='Pack Aggreg Camera Rig Sensor');	(**)

(*Single Input for PLAS*)

	st_I_MasterlistDoorGuard1				: ST_IO2_SingleInputCtrl:=			(eTypeInput:=NC,		tTimeOnFilter:=t#50ms, 		tTimeOffFilter:=t#50ms, 	sInputName:='Masterlist Door Guard1');	(**)
	st_I_MasterlistDoorGuard2				: ST_IO2_SingleInputCtrl:=			(eTypeInput:=NC,		tTimeOnFilter:=t#50ms, 		tTimeOffFilter:=t#50ms, 	sInputName:='Masterlist Door Guard2');	(**)
	st_I_MasterlistDoorGuard3				: ST_IO2_SingleInputCtrl:=			(eTypeInput:=NC,		tTimeOnFilter:=t#50ms, 		tTimeOffFilter:=t#50ms, 	sInputName:='Masterlist Door Guard3');	(**)

	st_I_OuterBrushOpen						: ST_IO2_SingleInputCtrl:=			(eTypeInput:=NC,		tTimeOnFilter:=t#50ms, 		tTimeOffFilter:=t#50ms, 	sInputName:='Outer Brush Open');	(**)
	st_I_PackAggregationDoorGuard1			: ST_IO2_SingleInputCtrl:=			(eTypeInput:=NC,		tTimeOnFilter:=t#50ms, 		tTimeOffFilter:=t#50ms, 	sInputName:='Pack Aggregation Door Guard1');	(**)
	st_I_PackAggregationDoorGuard2			: ST_IO2_SingleInputCtrl:=			(eTypeInput:=NC,		tTimeOnFilter:=t#50ms, 		tTimeOffFilter:=t#50ms, 	sInputName:='Pack Aggregation Door Guard2');	(**)

	st_I_WrapperDoorGuard1					:  ST_IO2_SingleInputCtrl:=			(eTypeInput:=NC,		tTimeOnFilter:=t#50ms, 		tTimeOffFilter:=t#50ms, 	sInputName:='Wrapper Door Guard1');	(**)
	st_I_WrapperDoorGuard2					: ST_IO2_SingleInputCtrl:=			(eTypeInput:=NC,		tTimeOnFilter:=t#50ms, 		tTimeOffFilter:=t#50ms, 	sInputName:='Wrapper Door Guard2');	(**)

	st_I_HeatTunelPackReject			: ST_IO2_SingleInputCtrl:=			(eTypeInput:=NO,		tTimeOnFilter:=t#50ms, 		tTimeOffFilter:=t#50ms, 	sInputName:='Heat Tunenel Pack Reject Sensor');	(**)
	st_I_WrapperPackReject				: ST_IO2_SingleInputCtrl:=			(eTypeInput:=NC,		tTimeOnFilter:=t#50ms, 		tTimeOffFilter:=t#50ms, 	sInputName:='Wrapper Pack Reject Sensor');	(**)
	st_I_WrapperPackReject2				: ST_IO2_SingleInputCtrl:=			(eTypeInput:=NC,		tTimeOnFilter:=t#50ms, 		tTimeOffFilter:=t#50ms, 	sInputName:='Wrapper Pack Reject 2 Sensor');	(**)
	st_I_WrapperOuterComplete			: ST_IO2_SingleInputCtrl:=			(eTypeInput:=NC,		tTimeOnFilter:=t#50ms, 		tTimeOffFilter:=t#50ms, 	sInputName:='Wrapper Pushing Arm Sensor');	(**)
	st_I_InhibitIntermediateCamera		: ST_IO2_SingleInputCtrl:=			(eTypeInput:=NC,		tTimeOnFilter:=t#50ms, 		tTimeOffFilter:=t#50ms, 	sInputName:='Inhibit Intermediate Camera');	(**)

(*Single Input for Laser*)
	st_I_CoderReady					: ST_IO2_SingleInputCtrl:=			(eTypeInput:=NO,		tTimeOnFilter:=t#100ms, 		tTimeOffFilter:=t#0ms, 	sInputName:='LASER - Ready');	(**)
	st_I_CoderBusy					: ST_IO2_SingleInputCtrl:=			(eTypeInput:=NO,		tTimeOnFilter:=t#100ms, 		tTimeOffFilter:=t#0ms, 	sInputName:='LASER - Busy');	(**)
	st_I_WrappingMaterialPresent		: ST_IO2_SingleInputCtrl:=			(eTypeInput:=NO,		tTimeOnFilter:=t#100ms, 		tTimeOffFilter:=t#0ms, 	sInputName:='LASER - WrapPresent');	(**)
	st_I_TabKnifeMoving				: ST_IO2_SingleInputCtrl:=			(eTypeInput:=NO,		tTimeOnFilter:=t#100ms, 		tTimeOffFilter:=t#0ms, 	sInputName:='LASER - TabKnife');	(**)


(*Double Input Config*)

	st_I_RowComplete						: ST_IO2_DoubleInputCtrl:=		(eInputSource:=SENSOR,	sInputName:='Row Complete',
																						eTypeInput1:=NO,		tTimeOnFilter1:=t#0ms,	tTimeOffFilter1	:=t#0ms,	(**)
											 											eTypeInput2:=NO,		tTimeOnFilter2:=t#0ms,	tTimeOffFilter2	:=t#0ms);	(**)
	st_I_LayerComplete					: ST_IO2_DoubleInputCtrl:=		(eInputSource:=SENSOR,	sInputName:='Layer Complete',
																						eTypeInput1:=NO,		tTimeOnFilter1:=t#0ms,	tTimeOffFilter1	:=t#0ms,	(**)
											 											eTypeInput2:=NO,		tTimeOnFilter2:=t#0ms,	tTimeOffFilter2	:=t#0ms);	(**)
	st_I_IntermediatePush					: ST_IO2_DoubleInputCtrl:=		(eInputSource:=SENSOR,	sInputName:='Intermediate Push',
																						eTypeInput1:=NO,		tTimeOnFilter1:=t#0ms,	tTimeOffFilter1	:=t#0ms,	(**)
											 											eTypeInput2:=NO,		tTimeOnFilter2:=t#0ms,	tTimeOffFilter2	:=t#0ms);	(**)
	st_I_CaseComplete					: ST_IO2_DoubleInputCtrl:=		(eInputSource:=SENSOR,	sInputName:='Case Complete',
																						eTypeInput1:=NO,		tTimeOnFilter1:=t#0ms,	tTimeOffFilter1	:=t#0ms,	(**)
											 											eTypeInput2:=NO,		tTimeOnFilter2:=t#0ms,	tTimeOffFilter2	:=t#0ms);	(**)
	st_I_CaseDischarged					: ST_IO2_DoubleInputCtrl:=		(eInputSource:=SENSOR,	sInputName:='Case Discharged',
																						eTypeInput1:=NO,		tTimeOnFilter1:=t#0ms,	tTimeOffFilter1	:=t#0ms,	(**)
											 											eTypeInput2:=NO,		tTimeOnFilter2:=t#0ms,	tTimeOffFilter2	:=t#0ms);	(**)
	st_I_CaseLabelValidation				: ST_IO2_DoubleInputCtrl:=		(eInputSource:=SENSOR,	sInputName:='Case Label Validation',
																						eTypeInput1:=NO,		tTimeOnFilter1:=t#0ms,	tTimeOffFilter1	:=t#0ms,	(**)
											 											eTypeInput2:=NO,		tTimeOnFilter2:=t#0ms,	tTimeOffFilter2	:=t#0ms);	(**)
(*
	st_I_LiftComplete						: ST_IO2_DoubleInputCtrl:=		(eInputSource:=SENSOR,		eTypeInput1:=NO,		tTimeOnFilter1:=t#0ms,	tTimeOffFilter1	:=t#0ms,	(**)
											 											eTypeInput2:=NO,		tTimeOnFilter2:=t#0ms,	tTimeOffFilter2	:=t#0ms);	(**)
	st_I_StackComplete					: ST_IO2_DoubleInputCtrl:=		(eInputSource:=SENSOR,		eTypeInput1:=NO,		tTimeOnFilter1:=t#0ms,	tTimeOffFilter1	:=t#0ms,	(**)
											 											eTypeInput2:=NO,		tTimeOnFilter2:=t#0ms,	tTimeOffFilter2	:=t#0ms);	(**)
	st_I_BundleCrossPushComplete		: ST_IO2_DoubleInputCtrl:=		(eInputSource:=SENSOR,		eTypeInput1:=NO,		tTimeOnFilter1:=t#0ms,	tTimeOffFilter1	:=t#0ms,	(**)
											 											eTypeInput2:=NO,		tTimeOnFilter2:=t#0ms,	tTimeOffFilter2	:=t#0ms);	(**)
	st_I_BundleTranferComplete			: ST_IO2_DoubleInputCtrl:=		(eInputSource:=SENSOR,		eTypeInput1:=NO,		tTimeOnFilter1:=t#0ms,	tTimeOffFilter1	:=t#0ms,	(**)
											 											eTypeInput2:=NO,		tTimeOnFilter2:=t#0ms,	tTimeOffFilter2	:=t#0ms);	(**)
*)


(*Output Config*)
	st_Q_TPDMachineRun					: ST_IO2_OutputCtrl:=			(eTypeOutput:=NO,		tOutputDelayed:=t#0ms,		tOutputLocked:=t#0ms,	sOutputName:='TPD Machine Run');		(* *)
	st_Q_CMLConvoyerRun				: ST_IO2_OutputCtrl:=			(eTypeOutput:=NO,		tOutputDelayed:=t#0ms,		tOutputLocked:=t#0ms,	sOutputName:='CML Convoyer Run');		(* *)
	st_Q_EUCAPreMachineRun				: ST_IO2_OutputCtrl:=			(eTypeOutput:=NO,		tOutputDelayed:=t#0ms,		tOutputLocked:=t#0ms,	sOutputName:='EUCA Machine Run');		(* *)
	st_Q_EUCAMachineRun				: ST_IO2_OutputCtrl:=			(eTypeOutput:=NO,		tOutputDelayed:=t#0ms,		tOutputLocked:=t#0ms,	sOutputName:='EUCA Machine Run');		(* *)
	st_Q_CaseContentOK					: ST_IO2_OutputCtrl:=			(eTypeOutput:=NO,		tOutputDelayed:=t#0ms,		tOutputLocked:=t#0ms,	sOutputName:='Case Content OK');		(* *)
	st_Q_CaseValidationOK				: ST_IO2_OutputCtrl:=			(eTypeOutput:=NO,		tOutputDelayed:=t#0ms,		tOutputLocked:=t#0ms,	sOutputName:='Case Validation OK');		(* *)
	st_Q_OuterValidationOK				: ST_IO2_OutputCtrl:=			(eTypeOutput:=NO,		tOutputDelayed:=t#0ms,		tOutputLocked:=t#0ms,	sOutputName:='Outer Validation OK');		(* *)
	st_Q_LabellerInhibit					: ST_IO2_OutputCtrl:=			(eTypeOutput:=NO,		tOutputDelayed:=t#0ms,		tOutputLocked:=t#0ms,	sOutputName:='Labeller Inhibit');		(* *)
	st_Q_SideBeltDriveBrake				: ST_IO2_OutputCtrl:=			(eTypeOutput:=NO,		tOutputDelayed:=t#500ms,	tOutputLocked:=t#20ms,	sOutputName:='Side Belt Drive Brake');		(* *)
	st_Q_PackSeparatorDriveBrake			: ST_IO2_OutputCtrl:=			(eTypeOutput:=NO,		tOutputDelayed:=t#200ms,	tOutputLocked:=t#100ms,sOutputName:='Pack Separator Drive Brake');		(* *)

	st_Q_CameraLightning1				: ST_IO2_OutputCtrl:=			(eTypeOutput:=NO,		tOutputDelayed:=t#0ms,		tOutputLocked:=t#15ms,	sOutputName:='Camera Lightning 1');		(* *)
	st_Q_CameraLightning2				: ST_IO2_OutputCtrl:=			(eTypeOutput:=NO,		tOutputDelayed:=t#0ms,		tOutputLocked:=t#15ms,	sOutputName:='Camera Lightning 2');		(* *)
	st_Q_CameraLightning3				: ST_IO2_OutputCtrl:=			(eTypeOutput:=NO,		tOutputDelayed:=t#0ms,		tOutputLocked:=t#15ms,	sOutputName:='Camera Lightning 3');		(* *)
	st_Q_CameraLightning4				: ST_IO2_OutputCtrl:=			(eTypeOutput:=NO,		tOutputDelayed:=t#0ms,		tOutputLocked:=t#15ms,	sOutputName:='Camera Lightning 4');		(* *)
	st_Q_CameraLightning5				: ST_IO2_OutputCtrl:=			(eTypeOutput:=NO,		tOutputDelayed:=t#0ms,		tOutputLocked:=t#15ms,	sOutputName:='Camera Lightning 5');		(* *)
	st_Q_CameraLightning6				: ST_IO2_OutputCtrl:=			(eTypeOutput:=NO,		tOutputDelayed:=t#0ms,		tOutputLocked:=t#15ms,	sOutputName:='Camera Lightning 6');		(* *)
	st_Q_CameraLightning7				: ST_IO2_OutputCtrl:=			(eTypeOutput:=NO,		tOutputDelayed:=t#0ms,		tOutputLocked:=t#15ms,	sOutputName:='Camera Lightning 7');		(* *)
	st_Q_CameraLightning8				: ST_IO2_OutputCtrl:=			(eTypeOutput:=NO,		tOutputDelayed:=t#0ms,		tOutputLocked:=t#15ms,	sOutputName:='Camera Lightning 8');		(* *)
	st_Q_CameraLightning9				: ST_IO2_OutputCtrl:=			(eTypeOutput:=NO,		tOutputDelayed:=t#0ms,		tOutputLocked:=t#15ms,	sOutputName:='Camera Lightning 9');		(* *)
	st_Q_CameraLightning10				: ST_IO2_OutputCtrl:=			(eTypeOutput:=NO,		tOutputDelayed:=t#0ms,		tOutputLocked:=t#15ms,	sOutputName:='Camera Lightning 10');	(* *)
	st_Q_CameraLightning11				: ST_IO2_OutputCtrl:=			(eTypeOutput:=NO,		tOutputDelayed:=t#0ms,		tOutputLocked:=t#15ms,	sOutputName:='Camera Lightning 11');	(* *)
	st_Q_CameraLightning12				: ST_IO2_OutputCtrl:=			(eTypeOutput:=NO,		tOutputDelayed:=t#0ms,		tOutputLocked:=t#15ms,	sOutputName:='Camera Lightning 12');	(* *)

(*Output Config for camera triggers*)
(*
	st_Q_Camera01						: ST_IO2_OutputCtrl:=			(eTypeOutput:=NO,		tOutputDelayed:=t#0ms,		tOutputLocked:=t#0ms);		(* *)
	st_Q_Camera02						: ST_IO2_OutputCtrl:=			(eTypeOutput:=NO,		tOutputDelayed:=t#0ms,		tOutputLocked:=t#0ms);		(* *)
	st_Q_Camera03						: ST_IO2_OutputCtrl:=			(eTypeOutput:=NO,		tOutputDelayed:=t#0ms,		tOutputLocked:=t#0ms);		(* *)
	st_Q_Camera04						: ST_IO2_OutputCtrl:=			(eTypeOutput:=NO,		tOutputDelayed:=t#0ms,		tOutputLocked:=t#0ms);		(* *)
	st_Q_Camera05						: ST_IO2_OutputCtrl:=			(eTypeOutput:=NO,		tOutputDelayed:=t#0ms,		tOutputLocked:=t#0ms);		(* *)
	st_Q_Camera06						: ST_IO2_OutputCtrl:=			(eTypeOutput:=NO,		tOutputDelayed:=t#0ms,		tOutputLocked:=t#0ms);		(* *)
	st_Q_Camera07						: ST_IO2_OutputCtrl:=			(eTypeOutput:=NO,		tOutputDelayed:=t#0ms,		tOutputLocked:=t#0ms);		(* *)
	st_Q_Camera08						: ST_IO2_OutputCtrl:=			(eTypeOutput:=NO,		tOutputDelayed:=t#0ms,		tOutputLocked:=t#0ms);		(* *)
	st_Q_Camera09						: ST_IO2_OutputCtrl:=			(eTypeOutput:=NO,		tOutputDelayed:=t#0ms,		tOutputLocked:=t#0ms);		(* *)
	st_Q_Camera10						: ST_IO2_OutputCtrl:=			(eTypeOutput:=NO,		tOutputDelayed:=t#0ms,		tOutputLocked:=t#0ms);		(* *)
	st_Q_Camera11						: ST_IO2_OutputCtrl:=			(eTypeOutput:=NO,		tOutputDelayed:=t#0ms,		tOutputLocked:=t#0ms);		(* *)
	st_Q_Camera12						: ST_IO2_OutputCtrl:=			(eTypeOutput:=NO,		tOutputDelayed:=t#0ms,		tOutputLocked:=t#0ms);		(* *)
*)
(******************************************************************************************************************************************************)

(*Shift Setup schedule*)
	aShiftSchedule									: ARRAY[1..cSHIFTNUMBER] OF TIMESTRUCT;
	aShiftChangeActive							: ARRAY[1..cSHIFTNUMBER] OF BOOL;

(*Pack*)
	tPackMasterListTimeout						: TIME := t#250ms;
	tPackAgreggationTimeout						: TIME := t#500ms;
	tPackConfirmationTimeout					: TIME := t#500ms;
	bCameraOnLeftSide							: BOOL; 	(*Set to true if the camera is on the left hand side of the conveyor as the packs travel trhough it towards the CML*)
	bPackCodesTrailing							: BOOL := TRUE; 	(*Set to true if the pack codes are on the trailing edge of the pack as it travels through the infeed cameras*)
	bFirstPackCodeOnTop							: BOOL;			(*Used for correct mapping packs from pack confirmation camera*)
	bDotCodeFormat								: BOOL;
	bQRCodeFormat								: BOOL;
	bEnableCodeAdjustment						: BOOL;
	bEnableCodeDuplicateCheck					: BOOL;
	nPacksPerStack								: UINT := 5;
	nMaxOutersBuffer								: UINT := 1; 		(*Maximum number of outers that can be processes at one time allowing for camera buffers - can be set higher if camera sequence max buffer is fixed!*)
	tBufferDelayTime								: TIME := t#200ms; 		(*Adjust this time so each outer stops for a moment before the first infeed camera sensor in order to avoid out of sync errors*)
	nConfirmationPackCode1						: INT := 1;
	nConfirmationPackCode2						: INT := 2;
	nCheckStatusOCV								: BYTE := 2;
	nExpectedValidationDepth						: INT:= 1;
	nInterimQueueIndex							: INT :=1;
	tInterimTimeout								: TIME := T#500ms;
	bLinearPackBufferExist							: BOOL;
	bExtendedOCVDupCheck						: BOOL;

	bEnableStopForInvalideCode					: BOOL;	(*Stop METS immidiatly after Lightbox detect invalide code*)
	bEnablePackCodeDateCheck					: BOOL;

	bFixedTriggerOffsetEnable						: BOOL;
	stPackAgregationCameraOffset				: ST_PACK_TriggerOffset;

	stPackCamera01Offset							: ST_PACK_TriggerOffset;
	stPackCamera02Offset							: ST_PACK_TriggerOffset;

(*Outer*)
	nOutersPerRow									: INT := 5;
	tTwoOutersOnRejectConv						:TIME := T#500ms;
	tRejectSensorTimeout							:TIME := T#2000ms;
	tOuterValidationTimeout						: TIME := t#750ms;
	bMasterListCameraDoubleRead				: BOOL := TRUE;
	nMasterListNumbersWarning					: INT := 5;
	bAggregationCameraRunWithTrigger			: BOOL;
	bAggregationStopOnInvalidCode				: BOOL ;
	bUseAuxRowCompleteSesnor					: BOOL;
	bUseInterimCodeForLastPosition				: BOOL;
	nAuxRowCount								: INT := 2;
	nAggregationQueueIndex						: INT :=0;
	tInspectionDelay								: TIME := t#30ms;
	bSkipStopGate									: BOOL;
	bPreLabelerShiftRegUsed						: BOOL;
	bConfirmOnOuter								: BOOL;
	bEanbleRestoreOCVFromConfirmation			: BOOL;
	bExtendedOACDupCheck						: BOOL;

(* Case*)
	nCaseQueueLength							: INT := 3;
	bPushIntoCaseCount							: BOOL;
	nCaseContentBuffer							: INT;
	bIntermediateBufferExist						: BOOL;
	bCasePackerDirectCutOut						: BOOL;
	bCasePositionOverwritingCheck				: BOOL := TRUE;
	tRowCompleteSignalTimeOut					: TIME := t#25s;
	tLayerCompleteSignalTimeOut					: TIME := t#25s;
	tIntermediatePushSignalTimeOut				: TIME := t#25s;
	tCaseCompleteSignalTimeOut					: TIME := t#25s;
	tDischargeSignalTimeOut						: TIME := t#25s;
	tCaseLabelValidationSignalTimeOut			: TIME := t#25s;
	bAddOACFromFileOnly						: BOOL;	(*Add OAC to infeed from file not from arrOuterStatus*)
	bSentOnlyGoodHierarchy						: BOOL := TRUE;
	bArchiveRejectedHierarchy					: BOOL := TRUE;
	bEnableStopOnOverWrittenData				: BOOL;
	bResetPushCountOnDoorOpen				: BOOL;
	bCheckDuplicateCaseLabel					: BOOL;
	bManualConfirmationEnable					: BOOL;
	bEnableStopOnCaseInavlid						: BOOL;
	bUseCaseFullAsValidationTrigger				: BOOL;
	bUseCaseContentReject						: BOOL;
	bUseRejectByCasepacker						: BOOL;
	tCaseRejectTimeOut							: TIME := t#60s;
	bAggregationWithoutCamera					: BOOL;
	bOrcaExist										: BOOL;

(*Archive settings*)
	nMaximumArchiveAge							: INT := 28;		(*Max archive age in days*)
	nMaximumArchiveFiles						: INT := 100;

	nMaximumOCVFiles							: INT := 5000;
	nMaximumOACFiles							: INT := 1000;
	nMaximumErrorFiles							: INT := 100;

(* HMI settings*)
	nWarningLevelPack							: REAL := 99.95;
	nAlarmLevelPack								: REAL := 99.9;
	nWarningLevelOuter							: REAL := 99.5;
	nAlarmLevelOuter								: REAL := 99.0;
	nWarningLevelCase							: REAL := 99.5;
	nAlarmLevelCase								: REAL := 95.0;

(* UPS Settings*)
	bUPSExist										: BOOL;
	tUPSShutdownDelay							: TIME := t#30s;		(*Default grace period for NT_Shutdown FB*)
	bUPSImmediateShutdown						: BOOL := FALSE;		(*Option to control immediate shutdown on power loss*)
END_STRUCT
END_TYPE

// ---- Global Variables/gMessage.TcGVL
{attribute 'qualified_only'}
{attribute 'Tc2GvlVarNames'}
VAR_GLOBAL

(************************************************************************************)

	aAlarms 			: ARRAY [0..cMAX_ALARM_GROUP] OF ST_Alarms;
	aAlarmsSettings 	: ARRAY [0..cMAX_ALARM_GROUP] OF ST_AlarmSettings;

	stAlarmTable		: ST_AlarmsTable;
	stAlarmStatus		: ST_AlarmStatus;
	
	
(**Alarms DWord releted to Infeed Case Packer Sequence**************)

	bAlarm_PackCodeDataInvalid					: BOOL;
	bAlarm_ConsecutivePackCodeDataInvalid		: BOOL;
	bAlarm_DuplicatePackCode					: BOOL;(*bAlarm_DuplicatePackCode*)

	bWarning_DuplicatePackCode					: BOOL;
	bWarning_DuplicateOCVRemoved				: BOOL;
	bWarning_OCVStackOutOfSequence				: BOOL;
	bAlarm_ConsecutiveOCVStackOutOfSeq			: BOOL;

	bWarning_OCVArmOutOfSequence				: BOOL;
	bWarning_OCVContentRepairing				: BOOL;
	bAlarm_ConsecutiveOCVMissing				: BOOL;

	bAlarm_ConsecutiveIntermediateNoRead		: BOOL;
	bAlarm_DuplicateIntermediateCode			: BOOL;

	bWarning_TwoOutersInAggregationArea			: BOOL; (*used in SFLX*)
	bAlarm_OuterAtChuteExitNotConfirmed			: BOOL;	(*used in SFLX*)
	bAlarm_OuterRejectNotConfirmed				: BOOL;
	bAlarm_OuterDataInvalide					: BOOL;
	bAlarm_ConsecutiveOuterRejects				: BOOL;
	bAlarm_DuplicateOuterLabel					: BOOL;
	bWarning_DuplicateOACRemoved				: BOOL;

	bAlarm_InfeedQueueInvalideData				: BOOL;
	bAlarm_InfeedQueueDuplicateData				: BOOL;
	bWarning_CaseContentMissing					: BOOL;(*bWarning_CaseContentMissing*)
	bAlarm_CaseContentNotFound					: BOOL;(*bAlarm_CaseContentNotFound*)
	bAlarm_ConsecutiveCaseContentMissing		: BOOL;(*bAlarm_ConsecutiveCaseContentMissing*)
	bAlarm_DuplicateCaseContentLabel			: BOOL; (*bAlarm_DuplicateCaseLabel*)
	bAlarm_CaseContentDataInvalide				: BOOL; (*bAlarm_CaseLabelInvalidData*)
	bWarrning_DuplicatesFoundInCase				: BOOL; (*stCaseQueue.stPrintCHMData.GenericHierarchy.CaseItem.RejectReason*)

	nAlarm_DataOverWrittenInCaseQueue			: BYTE;(*nAlarm_DataOverWrittenInCaseQueue*)

	bAlarm_CaseLabelInvalidData					: BOOL;
	bAlarm_ConsecutiveCaseRejects				: BOOL;
	bAlarm_DuplicateCaseLabel					: BOOL;
	nDuplicateCaseLabelIndex					: INT;
	bWarning_CaseReanimating					: BOOL;(*bWarning_CaseReanimating*)
	bWarning_OutersTooClose						: BOOL;

	(*bAlarm_CaseRejectedData				: BOOL;*)

(* *********************************************************** *)
(* *********           Printer alarms            	 ********* *)
(* *********************************************************** *)

	bAlarm_PrinterError				: BOOL;
	bAlarm_PritnerComms				: BOOL;

(* *********************************************************** *)
(* *********      Global DB Error  alarms flag       ********* *)
(* *********************************************************** *)

	bAlarm_AuxPCVCheckDBError			: BOOL;
	bAlarm_PCVCheckDBError				: BOOL;
	bAlarm_OCVCheckDBError				: BOOL;
	bAlarm_OACCheckDBError				: BOOL;
	bAlarm_OACCaseCheckDBError			: BOOL;
	bAlarm_CACCheckDBError				: BOOL;

(* *********************************************************** *)
(* *********           G03_EtherCAT alarms           ********* *)
(* *********************************************************** *)

	bAlarm_EtherCAT_IO_Error			: BOOL;

(* *********************************************************** *)
(* *********           NV memory overlap alarms           ********* *)
(* *********************************************************** *)

	nAlarm_OverlapNVMemCheck			: WORD;
	nAlarm_OverlapBitDisplay			: WORD;

END_VAR

// ---- Global Variables/gHMI.TcGVL
{attribute 'qualified_only'}
{attribute 'Tc2GvlVarNames'}
VAR_GLOBAL

	(*stPassthroughHMI 					: ST_HMI_Buttons;*)  (* - TO be replaced like in STG with status*)
	stVisualisation						: ST_HMI_Visualisation;

	stEnableForcingOutputs				: ST_HMI_Buttons;
	stForceOutputHMI					: ARRAY[1..6] OF ST_HMI_Buttons;

	nMachineStatusHMI					: INT;

	sPLCVersionHMI						: STRING;
	sPLCVersionInfoHMI					: T_MaxString;
	sPLCExternalInterfceHMI				: STRING;
	sScreenVersionInfoHMI				: T_MaxString;
	sBridgeVersionHMI					: STRING;

	(*nOuterSerialLenghtHMI				: UINT;	*)(*READ*)
	
	stStartHMI							: ST_HMI_Buttons;
	stStopHMI							: ST_HMI_Buttons;
	stResetHMI				 			: ST_HMI_Buttons;

	stResetTCPServerHMI					: ST_HMI_Buttons;

	aDebugDontStartScreenHMI			: ARRAY[1..2] OF ST_HMI_Buttons;
	stDebugDontStartBridgeHMI			: ST_HMI_Buttons;
    aWatchdogToHMI                      : ARRAY[1..cMAX_HMI_DISPLAYS] OF DINT;
    aWatchdogFromHMI                    : ARRAY[1..cMAX_HMI_DISPLAYS] OF DINT;

	stResetAllStatistics				: ST_HMI_Buttons;
	stResetPackInspectionHMI			: ST_HMI_Buttons;
	stResetOuterInspectionHMI			: ST_HMI_Buttons;
	stResetCaseInspectionHMI			: ST_HMI_Buttons;

	stResetAllCameraStatisticHMI		: ST_HMI_Buttons;

	stClearAlarmsWarningHistory			: ST_HMI_Buttons;

	stClearAllQueuesHMI					: ST_HMI_Buttons;
	stClearOuterArrayHMI				: ST_HMI_Buttons;
	stClearConveyorQueueHMI				: ST_HMI_Buttons;
	stClearPackerQueueHMI				: ST_HMI_Buttons;
	stClearCaseQueueHMI					: ST_HMI_Buttons;
	stClearOutfeedQueueHMI				: ST_HMI_Buttons;
	stClearCasePackerArrayHMI			: ST_HMI_Buttons;

	stClearVerifiedCaseDataHMI			: ST_HMI_Buttons;
	stClearFailedCaseDataHMI			: ST_HMI_Buttons;

	nClearDoneHMI						: WORD;

	aClearErrorDataHMI					: ARRAY[1..2] OF ST_HMI_Buttons;
	aErrorOuterPlusHMI					: ARRAY[1..2] OF ST_HMI_Buttons;
	aErrorOuterMinusHMI					: ARRAY[1..2] OF ST_HMI_Buttons;
	aErrorIndexHMI						: ARRAY[1..2] OF INT :=[2(1)];

	stForceNVClearHMI					: ST_HMI_Buttons;

	stManuallyReceivePCM				: ST_HMI_Buttons;
	(*nMEWebServiceStateHMI				: WORD;	(*READ BY PLC ONLY*) (*0-Created, 1 - Opening, 2 - Opened, 3 - Closing, 4 - Closed, 5 Faulted*)*)

	stShiftCSVStoreTable				: ST_HMI_CSVStoreTable;
	stProdCSVStoreTable					: ST_HMI_CSVStoreTable;

	(*HMI PLAS structure*)
	stPackLinearStatusHMI				: ST_HMI_PLAS_Queue;

	(*HMI PAOL structure*)
	stPackBufferStatusHMI				: ST_HMI_PACK_BufferStatus;

	(*sLastReadOuterBarcodeHMI			: T_OUTER_Barcode;
	aConfPackCodeInPositionHMI			: ARRAY[0..1] OF T_PACK_Barcode;*)
	stOuterAggregationHMI				: ST_HMI_OuterStatus;
	stFailureDiagnosticHMI				: ST_HMI_OuterStatus;
	bValidateForRejectDoneHMI			: BOOL;

	stInfeedConvQueueHMI				: ST_HMI_InfeedQueue;
	aPackerQueueHMI						: ARRAY [0..1] OF ST_HMI_InfeedQueue;

	aCaseQueueRejectCodeHMI				: ARRAY[1..cMAX_CASE_QUEUE] OF ST_HMI_CaseRejectCode;
	aVerifiedCaseIDCodeHMI				: ARRAY[1..cMAX_VERIFIED_CASE_QUEUE] OF ST_HMI_CaseVerifiedCode;
	aFailedCaseRejectCodeHMI			: ARRAY[1..cMAX_FAILED_CASE_QUEUE] OF ST_HMI_CaseRejectCode;

	(*CaseContent Aux data*)
	stCaseQueueHMI						: ST_HMI_CASE_CaseQueue;
	aFailedCACDataHMI					: ARRAY[1..cMAX_FAILED_CASE_QUEUE] OF ST_HMI_CAC_Data;	(* array of failed CAC data *)
	aVerifiedCACDataHMI					: ARRAY[1..cMAX_VERIFIED_CASE_QUEUE] OF ST_HMI_CAC_Data;	(* array of verified CAC data *)


	(*eTPDDriveStatusHMI				: E_HMI_DriveStatus;
	stLogAlarmsHMI						: ST_HMI_LogMessage;
	stLogWarrningsHMI					: ST_HMI_LogMessage;*)

	stBarGraph							: ST_HMI_BarGraph;
	bPerformanceTriggerHMI				: BOOL;
	bMemoRejectDoneForHMI				: BOOL;

(* Backup	 ************************************************************************************************)

	stCreateBackupHMI					: ST_HMI_Buttons;
	bBackupDoneHMI						: BOOL;
	sRestoreBackupNameHMI				: STRING;
	stRestoreBackupHMI					: ST_HMI_Buttons;
	bRestoreDoneHMI						: BOOL;

(* DB Report   ******************************************************************************************)

	stDBReportHMI						: ST_DB_ReportResult;

(* OLD CONTROL*)
	(*aAxisControlHMI					: ARRAY[1..cMAX_MC2_DRIVES] OF ST_HMI_AxisControl;*)

(* Manual Control ***************************************************************************************************)
	
	aCylinderCtrlHMI					: ARRAY[1..cMAX_CYLINDERS] OF ST_HMI_CylinderCtrl;
	aG120CtrlHMI						: ARRAY[1..cMAX_PROFINET_DRIVES] OF ST_HMI_G120Ctrl;
	aPrinterCtrlHMI						: ARRAY[1..cMAX_PRINTER_NUMBER] OF ST_HMI_PrinterCtrl;
	aAxisCtrlHMI						: ARRAY[1..cMAX_MC2_DRIVES] OF ST_HMI_AxisCtrl;

(* Device Status  ***************************************************************************************************)

	aCylinderStatusHMI					: ARRAY[1..cMAX_CYLINDERS] OF  ST_HMI_CylinderStatus;
	aG120StatusHMI						: ARRAY[1..cMAX_PROFINET_DRIVES] OF ST_HMI_G120Status;
	aPrinterStatusHMI					: ARRAY[1..cMAX_PRINTER_NUMBER] OF ST_HMI_PrinterStatus;
	aAxisStatusHMI						: ARRAY[1..cMAX_MC2_DRIVES] OF ST_HMI_AxisStatus;

	aHoneywellStatusHMI					: ARRAY[1..cMAX_HAND_SCANNERS] OF ST_HMI_HoneywellStatus;

(* HAND SCANNER ************************************************************************************************)

	stEnablePackInvalidSearchHMI		: ST_HMI_Buttons;

	bOCVSearchCodeHMI					: BOOL;
	sOCVSearchBarcodeHMI				: T_MaxString;
	stEnableInvalidOCVSearchHMI			: ST_HMI_Buttons;
	bOCVSearchCodeFoundHMI				: BOOL;

	bScanDoneHMI						: BOOL;
	sSearchedBarcodeHMI					: T_MaxString;
	stEnableOuterInvalidSearchHMI		: ST_HMI_Buttons;
	bOACSearchCodeFoundHMI				: BOOL;

	stEnablePackCodeRefeedHMI			: ST_HMI_Buttons;
	bRefeedButtonAvailableHMI			: BOOL;		(*bEnableRefeedButton*)

	stRemoveOuterFromQueueHMI			: ST_HMI_Buttons;
	stEnableCaseContentSearchHMI		: ST_HMI_Buttons;

(*
	bPackCodeFoundInDBHMI				:	 BOOL;	(*WRITE TO HMI ONLY*)
	bPackCodeNotFoundInDBHMI			: BOOL;	(*WRITE TO HMI ONLY*)
*)
	bRestoredOCVDataValidHMI			: BOOL;	(*WRITE TO HMI ONLY*)
	bRestoredOCVDataInvalidHMI			: BOOL;	(*WRITE TO HMI ONLY*)
	bRestoredOCVDataNotExistHMI			: BOOL;	(*WRITE TO HMI ONLY*)

	bRestoredOACDataValidHMI			: BOOL;	(*WRITE TO HMI ONLY*)
	bRestoredOACDataInvalidHMI			: BOOL;	(*WRITE TO HMI ONLY*)
	bRestoredOACDataNotExistHMI			: BOOL;	(*WRITE TO HMI ONLY*)

	bRestoredCACDataValidHMI			: BOOL;	(*WRITE TO HMI ONLY*)
	bRestoredCACDataInvalidHMI			: BOOL;	(*WRITE TO HMI ONLY*)
	bRestoredCACDataNotExistHMI			: BOOL;	(*WRITE TO HMI ONLY*)

	bRestoredCHMDataNotExistHMI			: BOOL;	(*WRITE TO HMI ONLY*)


(* CASE INSPACTION ************************************************************************************************)

	bCaseLabelScanCompleteHMI			: BOOL;	(*WRITE TO HMI ONLY*)

	(*outerinfeed conveyer *)
	nOuterProcessedHMI					: UDINT;
	nOuterAggregatedHMI					: UDINT;
	nMasterListRestoredSuccessfulHMI	: UDINT;	(*READ*)
	nMasterListRemovedHMI				: UDINT;	(*READ*)
	nQAButtonRejectOuterHMI				: UDINT;	(*READ*)

	(*row validation*)
	nRowValidationIndexUnderHMI			: UDINT;	(*READ*)
	nRowValidationIndexOverHMI			: UDINT;	(*READ*)
	nRowValidationIndexCorrectHMI		: UDINT;	(*READ*)
	nRowValidationIndexNotFoundHMI		: UDINT;	(*READ*)

	(*outer to case validation*)
	nOuterToCaseValidationIndexUnderHMI		: UDINT;	(*READ*)
	nOuterToCaseValidationIndexOverHMI		: UDINT;	(*READ*)
	nOuterToCaseValidationIndexCorrectHMI	: UDINT;	(*READ*)
	nOuterToCaseValidationIndexNoDataHMI	: UDINT;	(*READ*)

	(*case validation*)
	nCaseValidationScannedHMI				: UDINT;	(*READ*)
	nCaseValidationCorrectHMI				: UDINT;	(*READ*)
	nCaseValidationCasePackerRejectHMI		: UDINT;	(*READ*)
	nCaseValidationNoCaseLabelHMI			: UDINT;	(*READ*)

(* CASE PACKER SIGNALS  ******************************************************************************************)

	(*RowComplete*)
	nRowCompleteSensorHMI				: UDINT;	(*READ/WRITE*)
	nRowCompleteMachineHMI				: UDINT;	(*READ/WRITE*)
	nRowCompleteHMI						: UDINT;	(*READ/WRITE*)

	(*LayerComplete*)
	nLayerCompleteSensorHMI				: UDINT;	(*READ/WRITE*)
	nLayerCompleteMachineHMI			: UDINT;	(*READ/WRITE*)
	nLayerCompleteHMI					: UDINT;	(*READ/WRITE*)

	(*CaseComplete*)
	nCaseCompleteSensorHMI				: UDINT;	(*READ/WRITE*)
	nCaseCompleteMachineHMI				: UDINT;	(*READ/WRITE*)
	nCaseCompleteHMI					: UDINT;	(*READ/WRITE*)
	
	(*CaseComplete*)
	nCaseDischargedSensorHMI			: UDINT;	(*READ/WRITE*)
	nCaseDischargedMachineHMI			: UDINT;	(*READ/WRITE*)
	nCaseDischargedHMI					: UDINT;	(*READ/WRITE*)
	
	(*CaseLabelValidation*)
	nCaseLabelValidationSensorHMI		: UDINT;	(*READ/WRITE*)
	nCaseLabelValidationMachineHMI		: UDINT;	(*READ/WRITE*)
	nCaseLabelValidationHMI				: UDINT;	(*READ/WRITE*)


(* IO Status ******************************************************************************************************)

	aInputsStatusHMI					: ARRAY[1..64] OF ST_IO2_Diagnostic;
	aOutputsStatusHMI					: ARRAY[1..32] OF ST_IO2_Diagnostic;
	aForceOutputsHMI					: ARRAY[1..6] OF ST_IO2_Diagnostic;
	

END_VAR

// ---- Global Variables/InputsOutputsDT/gCamDevice.TcGVL
{attribute 'qualified_only'}
VAR_GLOBAL
	
	aCameraConfig	: ARRAY[1..2] OF ST_SCANNER_Configuration;
	aCameraStatus	: ARRAY[1..2] OF ST_SCANNER_Status;
	aCameraControl	: ARRAY[1..2] OF ST_SCANNER_Ctrl;
END_VAR

// ---- Global Variables/InputsOutputsDT/IOVarDT_S.TcGVL
{attribute 'Tc2GvlVarNames'}
VAR_GLOBAL
    bDT_TestErrorBypass								   : BOOL;	(* TRUE *)

	ibDT_24VPowerSupplyOK 						AT %I* : BOOL;	(* TRUE *)
	ibDT_PSRIsResetSignal						AT %I* : BOOL;	(* TRUE *)
	ibDT_PSRIsOkaySignal						AT %I* : BOOL;	(* TRUE *)
	ibDT_EmergencyStopFrom						AT %I* : BOOL;	(* TRUE *)
	ibDT_EmergancyCircuitSignal					AT %I* : BOOL;	(* TRUE *)

	ibDT_PreMachineInAutorun					AT %I* : BOOL;	(* TRUE *)
	ibDT_PostMachineInAutorun					AT %I* : BOOL;	(* TRUE *)
	ibDT_PackSeparationDriveOK					AT %I* : BOOL;	(* TRUE *)
	ibDT_PackIsolatorDrive						AT %I* : BOOL;	(* TRUE *)

	ibDT_PrePackAggregationCameraRigTrigger		AT %I* : BOOL;	(* SEQ *)
	ibDT_PackAggregationCamera1Trigger			AT %I* : BOOL;	(* SEQ *)
	ibDT_PackAggregationCamera2Trigger			AT %I* : BOOL;	(* SEQ *)
	ibDT_PackAggregationCamera3Trigger 			AT %I* : BOOL;	(* SEQ *)
	ibDT_PackAggregationCamera4Trigger 			AT %I* : BOOL;	(* For future *)

	ifDT_EncoderPosition						AT %I* : UDINT;
	ibDT_OuterValidationCameraTrigger			AT %I* : BOOL;	(* SEQ *)

	ibDT_RowCompleteSensor						AT %I* : BOOL;	(* DONE *)
	ibDT_LayerCompleteSensor					AT %I* : BOOL;	(* DONE *)
	ibDT_IntermediatePushSensor					AT %I* : BOOL;	(* For future *)
	ibDT_CaseCompleteSensor						AT %I* : BOOL;	(* DONE *)
	ibDT_CaseDischargedSensor					AT %I* : BOOL;	(* DONE *)
	ibDT_CaseLabelValidationTrigSensor 			AT %I* : BOOL;	(* DONE *)

	qbDT_PackAggregation01CameraTriggerOut		AT %Q* : BOOL;	(* SEQ *)
	qbDT_PackAggregation02CameraTriggerOut		AT %Q* : BOOL;	(* SEQ *)
	qbDT_PackAggregation03CameraTriggerOut		AT %Q* : BOOL;	(* SEQ *)

	qbDT_RearConfirmationCameraTriggerOut		AT %Q* : BOOL;
	qbDT_FrontConfirmationCameraTriggerOut		AT %Q* : BOOL;
	qbDT_OuterValidationCameraTriggerOut		AT %Q* : BOOL;

	qbDT_OuterAggregationCameraTriggerOut		AT %Q* : BOOL;
	qbDT_CaseContentValidationCameraTriggerOut 	AT %Q* : BOOL;
	qbDT_CaseLabelValidationCameraTriggerOut	AT %Q* : BOOL;
END_VAR

// ---- Global Variables/InputsOutputsDT/IOVarDT_H.TcGVL
VAR_GLOBAL
	
	(***************************Terminal States Diagnostic*****************************************************)

	istEtherCATMasterState								AT	%I*	: ST_CX_EtherCATMasterState;
	iaEtherCATSlaveState								AT 	%I*	: ARRAY [0..cMAX_ETHERCAT_SLAVES] OF UINT;

(*****************************Input/Output Cards*********************************************************)

	(*TERMINAL DTKF1 (EK1100 EtherCAT Power supply (2A E-Bus)) ***************************************)


	(*TERMINAL DT01KF1 (EL1008 8Ch. Dig. Input 24V, 3ms) ******************************************************)
	ibDT01KF1_1_EL1008									AT %I*: BOOL;
	ibDT01KF1_5_EL1008									AT %I*: BOOL;
	ibDT01KF1_2_EL1008									AT %I*: BOOL;
	ibDT01KF1_6_EL1008									AT %I*: BOOL;
	ibDT01KF1_3_EL1008 									AT %I*: BOOL;
	ibDT01KF1_7_EL1008									AT %I*: BOOL;
	ibDT01KF1_4_EL1008									AT %I*: BOOL;
	ibDT01KF1_8_EL1008 	 								AT %I*: BOOL;
	
	(*TERMINAL DT02KF1 (EL1008 8Ch. Dig. Input 24V, 3ms) ******************************************************)
	ibDT02KF1_1_EL1008									AT %I*: BOOL;
	ibDT02KF1_5_EL1008									AT %I*: BOOL;
	ibDT02KF1_2_EL1008									AT %I*: BOOL;
	ibDT02KF1_6_EL1008									AT %I*: BOOL;
	ibDT02KF1_3_EL1008 									AT %I*: BOOL;
	ibDT02KF1_7_EL1008									AT %I*: BOOL;
	ibDT02KF1_4_EL1008									AT %I*: BOOL;
	ibDT02KF1_8_EL1008	 								AT %I*: BOOL;
	
	(*TERMINAL DT03KF1 (EL2008 8Ch. Dig. Output 24V, 0.5A) ******************************************************)
	qbDT03KF1_1_EL2008									AT %Q*: BOOL;
	qbDT03KF1_5_EL2008									AT %Q*: BOOL;
	qbDT03KF1_2_EL2008									AT %Q*: BOOL;
	qbDT03KF1_6_EL2008									AT %Q*: BOOL;
	qbDT03KF1_3_EL2008									AT %Q*: BOOL;
	qbDT03KF1_7_EL2008									AT %Q*: BOOL;
	qbDT03KF1_4_EL2008									AT %Q*: BOOL;
	qbDT03KF1_8_EL2008									AT %Q*: BOOL;
	
	(*TERMINAL DT04KF1 (EL2624 4Ch. Relay Output, 125 V AC, 30 V DC, 0.5 A AC, 2 A DC)******************)
	qbDT04KF1_1_EL2624									AT %Q*: BOOL;
	qbDT04KF1_2_EL2624									AT %Q*: BOOL;
	qbDT04KF1_3_EL2624									AT %Q*: BOOL;
	qbDT04KF1_4_EL2624									AT %Q*: BOOL;
	
	(*TERMINAL DT05KF1 (EL6001 Interface (RS232))  ********1-Channel Serial Interface RS232***********************)
	ibDT05KF1_EL6001_PortNo								AT %I*: UINT;
	istDT05KF1_EL6001_COMPortDataIn						AT %I*: EL6InData22B;
	qstDT05KF1_EL6001_COMPortDataOut					AT %Q*: EL6OutData22B;
	
	(*TERMINAL DT06KF1 (EL9410 EtherCAT Power supply extension (2A E-Bus)) **************************************)

	ibDT06KF1_EL9410_UndervoltageEBus					AT%I*: BOOL;
	ibDT06KF1_EL9410_Undervoltage						AT%I*: BOOL;
	
	(*TERMINAL DT07KF1 (EL9505 Power supply terminal 5V) ***************5V Power Supplay***********************)

	ibDT07KF1_EL9505_PowerStatusOK						AT%I*: BOOL;
	ibDT07KF1_EL9505_PowerOverloaded					AT%I*: BOOL;
	
	
	
	
	(*TERMINAL DTKF2 (EK1100 EtherCAT Power supply (2A E-Bus)) ***********************************************)
	
	
	(*TERMINAL DT01KF2 (EL7031-0030 Stepper motor terminal, 24 VDC, 2.8 A, 2 analog inputs 0 – 10V) **********)
	ibDT01KF2_EL7031_Underrange_01						AT %I*: BOOL;
	ibDT01KF2_EL7031_Overrange_01						AT %I*: BOOL;
	
	ibDT01KF2_EL7031_Underrange_02						AT %I*: BOOL;
	ibDT01KF2_EL7031_Overrange_02						AT %I*: BOOL;
	
	refDT01KF2_EL7031_Axis								: AXIS_REF;
	
	(*TERMINAL DT02KF2 (EL6070 | License Key Terminal for TwinCAT 3.1) ***************************************)
	
	
	(*TERMINAL DT03KF2 (EL7031-0030 Stepper motor terminal, 24 VDC, 2.8 A, 2 analog inputs 0 – 10V) **********)
	ibDT03KF2_EL7031_Underrange_01						AT %I*: BOOL;
	ibDT03KF2_EL7031_Overrange_01						AT %I*: BOOL;
	
	ibDT03KF2_EL7031_Underrange_02						AT %I*: BOOL;
	ibDT03KF2_EL7031_Overrange_02						AT %I*: BOOL;
	
	refDT03KF2_EL7031_Axis								: AXIS_REF;
	
	
	(*TERMINAL DTKF3 (EK1818 EtherCAT coupler with digital inputs and outputs) ************************)
	ibDTKF3_1_EK1818									AT %I*: BOOL;
	ibDTKF3_2_EK1818									AT %I*: BOOL;
	ibDTKF3_3_EK1818									AT %I*: BOOL;
	ibDTKF3_4_EK1818									AT %I*: BOOL;
	ibDTKF3_5_EK1818									AT %I*: BOOL;
	ibDTKF3_6_EK1818									AT %I*: BOOL;
	ibDTKF3_7_EK1818									AT %I*: BOOL;
	ibDTKF3_8_EK1818									AT %I*: BOOL;
	
	qbDTKF3_1_EK1818									AT %Q*: BOOL;
	qbDTKF3_2_EK1818									AT %Q*: BOOL;
	qbDTKF3_3_EK1818									AT %Q*: BOOL;
	qbDTKF3_4_EK1818									AT %Q*: BOOL;
	
	(*TERMINAL DT01KF3 (EL7211-9014 | Servo Motor Terminals with OCT (One Cable Technology) and STO, 48 V DC) **********)
	
	refDTKF3_EL7211_Axis								: AXIS_REF;
	
	(*TERMINAL DT02KF3 (EL1918 | EtherCAT Terminal, 8-channel digital input, 24 V DC, TwinSAFE, TwinSAFE Logic) **********)
// 	ibDT02KF3_1_EL1918_Input							AT %I*: BOOL;
// 	ibDT02KF3_2_EL1918_Input							AT %I*: BOOL;
// 	ibDT02KF3_3_EL1918_Input							AT %I*: BOOL;
// 	ibDT02KF3_4_EL1918_Input							AT %I*: BOOL;
// 	ibDT02KF3_5_EL1918_Input							AT %I*: BOOL;
// 	ibDT02KF3_6_EL1918_Input							AT %I*: BOOL;
// 	ibDT02KF3_7_EL1918_Input							AT %I*: BOOL;
// 	ibDT02KF3_8_EL1918_Input							AT %I*: BOOL;
	
	(*TERMINAL DT03KF3 (EL3208 | 8-channel Analog Input Terminals, temperature, RTD (Pt100, Pt1000, ...) 16 bit *******************)
	qnDT03KF3_1_EL3208									AT %I*: INT; 
	qnDT03KF3_2_EL3208									AT %I*: INT; 
	qnDT03KF3_3_EL3208									AT %I*: INT; 
	qnDT03KF3_4_EL3208									AT %I*: INT; 
	qnDT03KF3_5_EL3208									AT %I*: INT; 
	qnDT03KF3_6_EL3208									AT %I*: INT; 
	qnDT03KF3_7_EL3208									AT %I*: INT; 
	qnDT03KF3_8_EL3208									AT %I*: INT; 
	
END_VAR

// ---- Global Variables/InputsOutputsDT/_Labs.TcGVL
VAR_GLOBAL

(*Here are variables\Structures\FB what are not taking part in the METS procces, but are under developing  for new feautes or new modules testing  *)

	(*cMAX_VALIDATION_ITEMS			: UINT :=10;*)

	stGS1_AI_Definition			: ST_GS1_AI_Definition;

	aGS1_AI : ARRAY[1..cNUMBER_DEFINED_AI_TYPES] OF ST_GS1_AI_Attributs;
	aGS1_Decode_AI : ARRAY[1..cNUMBER_DEFINED_AI_TYPES] OF ST_GS1_Decode_AI;

	stGS1CodeInfo_Pack							: ST_GS1_CodeInfo :=		(eCodeLvlType :=E_LEVEL1);
	stGS1CodeInfo_Outer						: ST_GS1_CodeInfo :=		(eCodeLvlType :=E_LEVEL2);
	stGS1CodeInfo_Case							: ST_GS1_CodeInfo :=		(eCodeLvlType :=E_LEVEL3);

	aGS1CodeInfo	: ARRAY[1..4] OF ST_GS1_CodeInfo :=[ (eCodeLvlType :=E_LEVEL1),(eCodeLvlType :=E_LEVEL2),(eCodeLvlType :=E_LEVEL3)];

	(*aCodeInfo		: ARRAY[0..3] OF ST_CodeInfo := (eCodeType :=E_PACK), (eCodeType :=E_OUTER),(eCodeType :=E_CASE), (eCodeType :=E_NONE);*)

	aGS1CodeInfo1	: ARRAY[1..4] OF INT :=[ 1,2, 3, 4] ;

	eLogName	: E_LOG_Handler;

	nTooLow : UDINT;
	diagIndex :DINT;
	diaglower: DINT;
	nTooHigh : UDINT;
	aLogBytesRecieved : ARRAY[1..100] OF DINT;


	aOuters 	: ARRAY[1..3] OF ST_LAB_OuterData;
	aLabCACData	: ST_CAC_Data;
	
	aOCVDataDB_LAB	: 	ST_DB_OCVDataCtrl;
	aOACDataDB_LAB	: 	ST_DB_OACDataCtrl;
	
	stDiagOCVDataDB				: ST_DB_OCVDataCtrl;
	stDaigOACDataDB				: ST_DB_OACDataCtrl;
	
	bTempBlockReadFromStruct		: BOOL;		{warning 'Overwirte Read From Struct'}
END_VAR

// ---- Global Variables/InputsOutputs_CML/IOVariablesCX_CML.TcGVL
{attribute 'Tc2GvlVarNames'}
VAR_GLOBAL
(***************************Terminal States Diagnostic********************************)

	istEtherCATMasterState					AT	%I*	: ST_CX_EtherCATMasterState;
	iaEtherCATSlaveState					AT 	%I*	: ARRAY [0..cMAX_ETHERCAT_SLAVES] OF UINT;

(*****************************Input/Output Cards***********************************)

(*CX - Main unit*)
	(*TERMINAL 46KF2 (EK1200-5000 EtherCAT Power supply (2A E-Bus)) *****************************************)

(*TERMINAL 50KF1 (EL6001 Interface (RS232))  ********1-Channel Serial Interface RS232*****************)
	(*ib50KF1_EL6001PortNo								AT%I*: UINT;
	ist50KF1_HandScannerCOMPortDataIn					AT%I*: EL6InData22B;
	qst50KF1_HandScannerCOMPortDataOut					AT%Q*: EL6OutData22B;*)

(*TERMINAL 60KF1 - EL1008 ******************************************************)
	ib60KF1_1_AirPressureOK 							AT %I* : BOOL; (* 60KF1_1 *)
	ib60KF1_5_24VSupplyOK								AT %I* : BOOL; (* 60KF1_5 *)
	ib60KF1_2_PSRIsResetSignal							AT %I* : BOOL; (* 60KF1_2 *)
	ib60KF1_6_PSRIsOkaySignal							AT %I* : BOOL; (* 60KF1_6 *)
	ib60KF1_3_EmergancyStopSignal						AT %I* : BOOL; (* 60KF1_3 *)
	ib60KF1_7_EmergancyCircuitSignal						AT %I* : BOOL; (* 60KF1_7 *)
	ib60KF1_4_NetworkOK								AT %I* : BOOL; (* 60KF1_4 *)
	ib60KF1_8_Spare									AT %I* : BOOL; (* 60KF1_8 *)

(*TERMINAL 80KF1 - EL2008 ******************************************************)
	qb80KF1_1_SafetyResetSignal							AT %Q* : BOOL; (* 80KF1_1 *)
	qb80KF1_5_AdditionalSafetyResetSignal					AT %Q* : BOOL; (* 80KF1_5 *)
	qb80KF1_2_Spare									AT %Q* : BOOL; (* 80KF1_2 *)
	qb80KF1_6_Spare									AT %Q* : BOOL; (* 80KF1_6 *)
	qb80KF1_3_Spare									AT %Q* : BOOL; (* 80KF1_3 *)
	qb80KF1_7_Spare									AT %Q* : BOOL; (* 80KF1_7 *)
	qb80KF1_4_Spare									AT %Q* : BOOL; (* 80KF1_4 *)
	qb80KF1_8_Spare									AT %Q* : BOOL; (* 80KF1_8 *)

(*TERMINAL 95KF1 - EL6631 -  PROFINET IO Controller **************************************************)

	ist95KF1_Master01PNetState 							AT %I* : ST_CX_EtherCATMasterPNetState;

	(*DRIVE  403T1  - G120C *************************************************************************)
	ist403T1_infeedconveyor								AT %I* : ST_DRIVE_INPUT;
	qst403T1_infeedconveyor								AT %Q* : ST_DRIVE_OUTPUT;

	(*DRIVE  405T1  - G120C *************************************************************************)
	ist405T1_loweratorbelts								AT %I* : ST_DRIVE_INPUT;
	qst405T1_loweratorbelts								AT %Q* : ST_DRIVE_OUTPUT;

(*DRIVE  406T1  - G120C ******************************************************************************)
	ist406T1_rotarytransfer								AT %I* : ST_DRIVE_INPUT;
	qst406T1_rotarytransfer								AT %Q* : ST_DRIVE_OUTPUT;

(*DRIVE  407T1  - G120C ******************************************************************************)
	ist407T1_rejectconveyor								AT %I* : ST_DRIVE_INPUT;
	qst407T1_rejectconveyor								AT %Q* : ST_DRIVE_OUTPUT;

(*DRIVE  408T1  - G120C ******************************************************************************)
	ist408T1_slowdownmotors							AT %I* : ST_DRIVE_INPUT;
	qst408T1_slowdownmotors							AT %Q* : ST_DRIVE_OUTPUT;

(*DIS inputs 46KF2 (CX2100 Power Supply) ******************************************)

	ib446KF2_Up						 				AT %I* : BOOL;
	ib446KF2_Down		 							AT %I* : BOOL;
	ib446KF2_Left		 								AT %I* : BOOL;
	ib446KF2_Right	 									AT %I* : BOOL;
	ib446KF2_Enter	 									AT %I* : BOOL;

(*METS CML*)
	(*TERMINAL 446KF2 (EK1200-5000 EtherCAT Power supply (2A E-Bus)) *****************************************)

(*TERMINAL447KF1 (EL9410 E-Bus Power Supplier  (Diagnostics)) ***************2A Bus Supplay***********************)

	ib447KF1_UndervoltageUs							AT%I* : BOOL;
	ib447KF1_UndervoltageUp							AT%I* : BOOL;

(*TERMINAL 460KF1 - EL1008 ***********************************************************************)
	ib460KF1_1_Guard1UpperSideAccessDoor				AT %I* : BOOL; (* 460KF1_1 *)
	ib460KF1_5_Guard2UpperDoorLabellerSide				AT %I* : BOOL; (* 460KF1_5 *)
	ib460KF1_2_Guard3OutfeedTunnel						AT %I* : BOOL; (* 460KF1_2 *)
	ib460KF1_6_Guard4ElectricalBoxInPosition				AT %I* : BOOL; (* 460KF1_6 *)
	ib460KF1_3_Guard5RejectBinLHSide						AT %I* : BOOL; (* 460KF1_3 *)
	ib460KF1_7_Guard6RejectBinRHSide						AT %I* : BOOL; (* 460KF1_7 *)
	ib460KF1_4_Guard7HTTDoorGuard						AT %I* : BOOL; (* 460KF1_4 *)
	ib460KF1_8_Spare									AT %I* : BOOL; (* 460KF1_8 *)

(*TERMINAL 461KF1 - EL1008 ***********************************************************************)
	ib461KF1_1_Guard8Labeller1InPosition					AT %I* : BOOL; (* 461KF1_1 *)
	ib461KF1_5_Guard9Labeller2InPosition					AT %I* : BOOL; (* 461KF1_5 *)
	ib461KF1_2_Guard10FrontUpperDoor					AT %I* : BOOL; (* 461KF1_2 *)
	ib461KF1_6_Guard11GuardLowerLabellerSide				AT %I* : BOOL; (* 461KF1_6 *)
	ib461KF1_3_RejectBinGuardIsReset						AT %I* : BOOL; (* 461KF1_3 *)
	ib461KF1_7_Labeller1GuardIsReset						AT %I* : BOOL; (* 461KF1_7 *)
	ib461KF1_4_Labeller2GuardIsReset						AT %I* : BOOL; (* 461KF1_4 *)
	ib461KF1_8_Spare									AT %I* : BOOL; (* 461KF1_8 *)

(*TERMINAL 462KF1 - EL1008 ***********************************************************************)
	ib462KF1_1_Labeller1Ready							AT %I* : BOOL; (* 462KF1_1 *)
	ib462KF1_5_Labeller1SummaryWarning					AT %I* : BOOL; (* 462KF1_5 *)
	ib462KF1_2_FrontCameraTrigger						AT %I* : BOOL; (* 462KF1_2 *)
	ib462KF1_6_Labeller1DataReady						AT %I* : BOOL; (* 462KF1_6 *)
	ib462KF1_3_Labeller1HomePosition						AT %I* : BOOL; (* 462KF1_3 *)
	ib462KF1_7_Labeller1LabelPrinted						AT %I* : BOOL; (* 462KF1_7 *)
	ib462KF1_4_Labeller1Error							AT %I* : BOOL; (* 462KF1_4 *)
	ib462KF1_8_Labeller1OuterAtLabeller					AT %I* : BOOL; (* 462KF1_8 *)

(*TERMINAL 463KF1 - EL1008 ***********************************************************************)
	ib463KF1_1_Labeller2Ready							AT %I* : BOOL; (*4 63KF1_1 *)
	ib463KF1_5_Labeller2SummaryWarning					AT %I* : BOOL; (* 463KF1_5 *)
	ib463KF1_2_RearCameraTrigger							AT %I* : BOOL; (* 463KF1_2 *)
	ib463KF1_6_Labeller2DataReady						AT %I* : BOOL; (* 463KF1_6 *)
	ib463KF1_3_Lebeller2HomePosition						AT %I* : BOOL; (* 463KF1_3 *)
	ib463KF1_7_Labeller2LabelPrinted						AT %I* : BOOL; (* 463KF1_7 *)
	ib463KF1_4_Labeller2Error							AT %I* : BOOL; (* 463KF1_4 *)
	ib463KF1_8_Labeller2OuterAtLabeller					AT %I* : BOOL; (* 463KF1_8 *)

(*TERMINAL 464KF1 - EL1008 ***********************************************************************)
	ib464KF1_1_RotaryTransferPackAtStopPlate				AT %I* : BOOL; (* 464KF1_1 *)
	ib464KF1_5_RotaryTransferTorqueLimiter					AT %I* : BOOL; (* 464KF1_5 *)
	ib464KF1_2_RotaryTransferDelayStop1					AT %I* : BOOL; (* 464KF1_2 *)
	ib464KF1_6_RotaryTransferDelayStop2					AT %I* : BOOL; (* 464KF1_6 *)
	ib464KF1_3_Spare									AT %I* : BOOL; (* 464KF1_3 *)
	ib464KF1_7_Spare									AT %I* : BOOL; (* 464KF1_7 *)
	ib464KF1_4_Spare									AT %I* : BOOL; (* 464KF1_4 *)
	ib464KF1_8_Spare									AT %I* : BOOL; (* 464KF1_8 *)

(*TERMINAL 465KF1 - EL1008***********************************************************************)
	ib465KF1_1_OuterAtReject							AT %I* : BOOL; (* 465KF1_1 *)
	ib465KF1_5_CMLExitBlock								AT %I* : BOOL; (* 465KF1_5 *)
	ib465KF1_2_RejectPB								AT %I* : BOOL; (* 465KF1_2 *)
	ib465KF1_6_LoweratorGuideRHLowerInPosition			AT %I* : BOOL; (* 465KF1_6 *)
	ib465KF1_3_LoweratorGuideLHLowerInPosition			AT %I* : BOOL; (* 465KF1_3 *)
	ib465KF1_7_RejectCylinderExtended					AT %I* : BOOL; (* 465KF1_7 *)
	ib465KF1_4_RejectCylinderRetracted					AT %I* : BOOL; (* 465KF1_4 *)
	ib465KF1_8_RejectBinFull								AT %I* : BOOL; (* 465KF1_8 *)

(*TERMINAL 466KF1 - EL1008***********************************************************************)
	ib466KF1_1_AdditionalConveyor1Isolator					AT %I* : BOOL; (* 466KF1_1 *)
	ib466KF1_5_AdditionalConveyor2Isolator					AT %I* : BOOL; (* 466KF1_5 *)
	ib466KF1_2_AdditionalConveyor3Isolator					AT %I* : BOOL; (* 466KF1_2 *)
	ib466KF1_6_AdditionalConveyor4ThermalOverload			AT %I* : BOOL; (* 466KF1_6 *)
	ib466KF1_3_PreLabelCameraTrigger						AT %I* : BOOL; (* 466KF1_3 *)						(*not used on C922 and C925 *)
	ib466KF1_7_PostLabelCameraTrigger					AT %I* : BOOL; (* 466KF1_7 *)						(*not used on C922 and C925 *)
	ib466KF1_4_NCWShiftRegister							AT %I* : BOOL; (* 466KF1_4 *)						(*not used on C922 and C925 *)
	ib466KF1_8_ResetPB									AT %I* : BOOL; (* 466KF1_8 *)

(*TERMINAL 467KF1 - EL1008***********************************************************************)
	ib467KF1_1_Spare									AT %I* : BOOL; (* 467KF1_1 *)
	ib467KF1_5_OutfeedCleatedConveyorTorqueLimiter		AT %I* : BOOL; (* 467KF1_5 not used *)
	ib467KF1_2_AdditionalConveyor4OK					AT %I* : BOOL; (* 467KF1_2 sofstart is happy*)
	ib467KF1_6_Spare									AT %I* : BOOL; (* 467KF1_6 *)
	ib467KF1_3_PreMachineAutorun						AT %I* : BOOL; (* 467KF1_3 *)
	ib467KF1_7_PostMachineAutorun						AT %I* : BOOL; (* 467KF1_7 *)
	ib467KF1_4_ConveyorIndexContact						AT %I* : BOOL; (* 467KF1_4 delay stop for inffed conv for packs *)
	ib467KF1_8_OutfeedCleatedConveyorTransfer				AT %I* : BOOL; (* 467KF1_8 not used *)

(*TERMINAL 468KF1 - EL1008************************************************************************)
	ib468KF1_1_HTTMinimumLevel						AT %I* : BOOL; (* 468KF1_1 *)
	ib468KF1_5_HTTDatumSwich							AT %I* : BOOL; (* 468KF1_5 *)
	ib468KF1_2_HTTPackAtStop							AT %I* : BOOL; (* 468KF1_2 *)
	ib468KF1_6_HTTPackExitBlocked						AT %I* : BOOL; (* 468KF1_6 *)
	ib468KF1_3_HTTGuideCylinderExtended					AT %I* : BOOL; (* 468KF1_3 *)
	ib468KF1_7_PackBuildBackPreMachineCutout				AT %I* : BOOL; (* 468KF1_7 *)
	ib468KF1_4_InfeedCleatedConveyorTorqueLimiter			AT %I* : BOOL; (* 468KF1_4 *)
	ib468KF1_8_InfeedCleatedConveyorTransfer				AT %I* : BOOL; (* 468KF1_8 *)

(*TERMINAL 469KF1 - EL1008************************************************************************)
	ib469KF1_1_HTT2MinimumLevel						AT %I* : BOOL; (* 469KF1_1 *)						(*not used on C922 and C925 *)
	ib469KF1_5_HTT2DatumSwich							AT %I* : BOOL; (* 469KF1_5 *)						(*not used on C922 and C925 *)
	ib469KF1_2_HTT2PackAtStop							AT %I* : BOOL; (* 469KF1_2 *)						(*not used on C922 and C925 *)
	ib469KF1_6_HTT2ExitBlocked							AT %I* : BOOL; (* 469KF1_6 *)						(*not used on C922 and C925 *)
	ib469KF1_3_HTT2GuideCylinderExtended					AT %I* : BOOL; (* 469KF1_3 *)						(*not used on C922 and C925 *)
	ib469KF1_7_PackBuildBack2PreMachineCutout				AT %I* : BOOL; (* 469KF1_7 *)						(*not used on C922 and C925 *)
	ib469KF1_4_PreMachineHTT2ConveyorRun				AT %I* : BOOL; (* 469KF1_4 *)						(*not used on C922 and C925 *)
	ib469KF1_8_Spare									AT %I* : BOOL; (* 469KF1_8 *)						(*not used on C922 and C925 *)

(*TERMINAL 480KF1 - EL2008 ************************************************************************)
	qb480KF1_1_Spare									AT %Q* : BOOL; (* 480KF1_1 *)
	qb480KF1_5_AdditionalConveyor1Run					AT %Q* : BOOL; (* 480KF1_5 *)
	qb480KF1_2_AdditionalConveyor2Run					AT %Q* : BOOL; (* 480KF1_2 *)
	qb480KF1_6_AdditionalConveyor3Run					AT %Q* : BOOL; (* 480KF1_6 *)
	qb480KF1_3_AdditionalConveyor4Run					AT %Q* : BOOL; (* 480KF1_3 *)
	qb480KF1_7_Spare									AT %Q* : BOOL; (* 480KF1_7 *)
	qb480KF1_4_CleatedConveyrBrake						AT %Q* : BOOL; (* 480KF1_4 *)
	qb480KF1_8_PackSeparationMotorBrake					AT %Q* : BOOL; (* 480KF1_8 *)

(*TERMINAL 481KF1 - EL2008 ************************************************************************)
	qb481KF1_1_RejectCylinderExtend						AT %Q* : BOOL; (* 481KF1_1 *)	(*Solenoid*)
	qb481KF1_5_RejectCylinderRetract						AT %Q* : BOOL; (* 481KF1_5 *)	(*Solenoid*)
	qb481KF1_2_FrontHightResCameraPower					AT %Q* : BOOL; (* 481KF1_2 *)
	qb481KF1_6_ReartHightResCameraPower					AT %Q* : BOOL; (* 481KF1_6 *)
	qb481KF1_3_HTTGiudesCylinderExtend					AT %Q* : BOOL; (* 481KF1_3 *)	(*Solenoid*)
	qb481KF1_7_HTTGiudesCylinderRetract					AT %Q* : BOOL; (* 481KF1_7 *)	(*Solenoid*)
	qb481KF1_4_FrontHightResCameraTrigger				AT %Q* : BOOL; (* 481KF1_4 *)
	qb481KF1_8_ReartHightResCameraTrigger				AT %Q* : BOOL; (* 481KF1_8 *)

(*TERMINAL 482KF1 - EL2008 ************************************************************************)
	qb482KF1_1_RejectCameraPower						AT %Q*  : BOOL; (* 482KF1_1 *)	(*MasterListCameraPower*)
	qb482KF1_5_RejectCameraTrigger						AT %Q*  : BOOL; (* 482KF1_5 *)	(*MasterListCameraTrigger*)
	qb482KF1_2_PreLabelCameraPower						AT %Q*  : BOOL; (* 482KF1_2 *)						(*not used on C922 and C925 *)
	qb482KF1_6_PreLabelCameraTrigger						AT %Q*  : BOOL; (* 482KF1_6 *)						(*not used on C922 and C925 *)
	qb482KF1_3_PostLabelCameraPower					AT %Q*  : BOOL; (* 482KF1_3 *)						(*not used on C922 and C925 *)
	qb482KF1_7_PostLabelCameraTrigger					AT %Q*  : BOOL; (* 482KF1_7 *)						(*not used on C922 and C925 *)
	qb482KF1_4_Labbeller1ApplyAvailable					AT %Q*  : BOOL; (* 482KF1_4 *)
	qb482KF1_8_Labbeller2ApplyAvailable					AT %Q*  : BOOL; (* 482KF1_8 *)

(*TERMINAL 483KF1 - EL2008 ************************************************************************)
	qb483KF1_1_LightPoleGreen							AT %Q*  : BOOL; (* 483KF1_1 *)	(*MasterListCameraPower*)
	qb483KF1_5_LightPoleAmber							AT %Q*  : BOOL; (* 483KF1_5 *)	(*MasterListCameraTrigger*)
	qb483KF1_2_LightPoleRed							AT %Q*  : BOOL; (* 483KF1_2 *)
	qb483KF1_6_LightPoleAlarm							AT %Q*  : BOOL; (* 483KF1_6 *)
	qb483KF1_3_ResetPB								AT %Q*  : BOOL; (* 483KF1_3 *)
	qb483KF1_7_AdditionalPreMachineCutoutBeltInMotion		AT %Q*  : BOOL; (* 483KF1_7 *)
	qb483KF1_4_PreMachineCutoutSignalRelay				AT %Q*  : BOOL; (* 483KF1_4 *)
	qb483KF1_8_MachineRunSignalRelay					AT %Q*  : BOOL; (* 483KF1_8 *)

(*TERMINAL 490KF1 - EL2624 ************************************************************************)
	qb490KF1_1_Labeller1ResetSignal						AT %Q*  : BOOL; (*490KF1_1*)
	qb490KF1_2_Labeller2ResetSignal						AT %Q*  : BOOL; (*490KF1_2*)
	qb490KF1_3_Labeller1PrintSignal						AT %Q*  : BOOL; (*490KF1_3*)
	qb490KF1_4_Labeller2PrintSignal						AT %Q*  : BOOL; (*490KF1_4*)



END_VAR

// ---- Global Variables/InputsOutputs_CML/IOVariablesEUCA_CML.TcGVL
{attribute 'Tc2GvlVarNames'}
VAR_GLOBAL

(*****************************Input/Output Cards***********************************)

(*METS EUCA (CML)*)
	(*TERMINAL 646KF2 (EK1200-5000 EtherCAT Power supply (2A E-Bus)) *****************************************)

	ib650KF1_EL6001PortNo								AT%I*: UINT;
	ist650KF1_HandScannerCOMPortDataIn					AT%I*: EL6InData22B;
	qst650KF1_HandScannerCOMPortDataOut				AT%Q*: EL6OutData22B;

(*TERMINAL 651KF1 - EL4002 ******************************************************)
	qn651KF1_1_LightingIntensityOuterValidCamera			AT %Q* : INT;
	qn651KF1_2_LightingIntensityOuterAggCamera			AT %Q* : INT;

(*TERMINAL 652KF1 - EL4002 ******************************************************)
	qn652KF1_1_LightingIntensityCaseContentCamera		AT %Q* : INT;
	qn652KF1_2_Spare											AT %Q* : INT;

(*TERMINAL 660KF1 (EL1008 **************************************************************)
	ib660KF1_1_IntermediatePushSensor 					AT %I*: BOOL;(* 660KF1_1 *)
	ib660KF1_5_RowCompleteSensor 						AT %I*: BOOL;(* 660KF1_1 *)
	ib660KF1_2_LayerCompleteSensor 						AT %I*: BOOL;(* 660KF1_1 *)
	ib660KF1_6_CaseCompleteSensor 						AT %I*: BOOL;(* 660KF1_1 *)
	ib660KF1_3_CaseDischargedSensor 						AT %I*: BOOL;(* 660KF1_1 *)
	ib660KF1_7_Spare  									AT %I*: BOOL;(* 660KF1_1 *)
	ib660KF1_4_CaseLabelValidationTrigSensor				AT %I*: BOOL;(* 660KF1_1 *)
	ib660KF1_8_CaseLabelValidationTrig_SFCP 				AT %I*: BOOL;(* 660KF1_1 *)

(*TERMINAL 661KF1 (EL1008  **************************************************************)
	ib661KF1_1_DoorOpenZone1 							AT %I*: BOOL;(* 661KF1_1 *)
	ib661KF1_5_DoorOpenZone2 							AT %I*: BOOL;(* 661KF1_1 *)
	ib661KF1_2_CasePackerAutoRun_SFCP					AT %I*: BOOL;(* 661KF1_1 *)
	ib661KF1_6_CaseRejectet_SFCP 						AT %I*: BOOL;(* 661KF1_1 *)
	ib661KF1_3_RowComplete_SFCP 						AT %I*: BOOL;(* 661KF1_1 *)
	ib661KF1_7_LayerComplete_SFCP 						AT %I*: BOOL;(* 661KF1_1 *)
	ib661KF1_4_CaseComplete_SFCP 						AT %I*: BOOL;(* 661KF1_1 *)
	ib661KF1_8_CaseDischarged_SFCP 						AT %I*: BOOL;(* 661KF1_1 *)

(*TERMINAL 662KF1 (EL1008 **************************************************************)
	ib662KF1_1_24VSupplyOkay 							AT %I*: BOOL;(* 662KF1_1 *)
	ib662KF1_5_24VSupplyOkayAdditionalSupplySpare 			AT %I*: BOOL;(* 662KF1_1 *)
	ib662KF1_2_Spare 									AT %I*: BOOL;(* 662KF1_1 *)
	ib662KF1_6_Spare 									AT %I*: BOOL;(* 662KF1_1 *)
	ib662KF1_3_IntermediatePush_SFCP 					AT %I*: BOOL;(* 662KF1_1 *)
	ib662KF1_7_AdditionalPreMachineAutorun 				AT %I*: BOOL;(* 662KF1_1 *)					(*not used on C922 and C925 *)
	ib662KF1_4_Spare 									AT %I*: BOOL;(* 662KF1_1 *)
	ib662KF1_8_Spare			 						AT %I*: BOOL;(* 662KF1_1 *)

(*TERMINAL 680KF1 (EL2008  **************************************************************)
	qb680KF1_1_OuterMasterListCamTrig 					AT %Q*: BOOL;(* 680KF1_1 *)					(*not used on C922 and C925 *)		(*rejectCamera instead*)
	qb680KF1_5_OuterAggregationCamTrig 					AT %Q*: BOOL;(* 680KF1_1 *)
	qb680KF1_2_CaseContentValidationCamTrig   				AT %Q*: BOOL;(* 680KF1_1 *)
	qb680KF1_6_CaseLabelValidationCamTrig 				AT %Q*: BOOL;(* 680KF1_1 *)
	qb680KF1_3_OuterMasterListCameraPower  				AT %Q*: BOOL;(* 680KF1_1 *)					(*not used on C922 and C925 *)		(*rejectCamera instead*)	(*qb482KF1_1_RejectCameraPower*)
	qb680KF1_7_OuterAggregationCamPower  				AT %Q*: BOOL;(* 680KF1_1 *)
	qb680KF1_4_CaseContentValidationCamPower  			AT %Q*: BOOL;(* 680KF1_1 *)
	qb680KF1_8_CaseLabelValidationCamPower  				AT %Q*: BOOL;(* 680KF1_1 *)

(*TERMINAL 681KF1 (EL2008  **************************************************************)
	qb681KF1_1_Cutout_STCP  							AT %Q*: BOOL;(* 681KF1_1 *)
	qb681KF1_5_CaseValidationOK_STCP  					AT %Q*: BOOL;(* 681KF1_1 *)
	qb681KF1_2_OuterValidationOK_STCP  					AT %Q*: BOOL;(* 681KF1_1 *)
	qb681KF1_6_CaseContentOK_STCP						AT %Q*: BOOL;(* 681KF1_1 *)					(*not used on C922 and C925 *)
	qb681KF1_3_HandScannerLightPoleGreen 				AT %Q*: BOOL;(* 681KF1_1 *)
	qb681KF1_7_HandScannerLightPoleRed  					AT %Q*: BOOL;(* 681KF1_1 *)
	qb681KF1_4_Spare  									AT %Q*: BOOL;(* 681KF1_1 *)
	qb681KF1_8_CMLConvoyerRun   						AT %Q*: BOOL;(* 681KF1_1 *)(*OuterRejetcSignal*)	(*not used on C922 and C925 *)

(*TERMINAL 682KF1 (EL2008  **************************************************************)
	qb682KF1_1_Spare 										AT %Q*: BOOL;(* 682KF1_1 *)
	qb682KF1_5_Spare  										AT %Q*: BOOL;(* 682KF1_1 *)
	qb682KF1_2_Spare  										AT %Q*: BOOL;(* 682KF1_1 *)
	qb682KF1_6_Spare											AT %Q*: BOOL;(* 682KF1_1 *)
	qb682KF1_3_PLCControlledOuterValidCamLightning		AT %Q*: BOOL;(* 682KF1_1 *)
	qb682KF1_7_PLCControlledOuterAggCamLightning		AT %Q*: BOOL;(* 682KF1_1 *)
	qb682KF1_4_PLCControlledCaseContentCamLightning  	AT %Q*: BOOL;(* 682KF1_1 *)
	qb682KF1_8_Spare   										AT %Q*: BOOL;(* 682KF1_1 *)

(*TERMINAL 690KF1 (EL9505 Power supply terminal 5V) ***************5V Power Supplay***********************)

	ib690KF1_PowerStatusOK								AT%I* : BOOL;
	ib690KF1_PowerOverloaded							AT%I* : BOOL;

END_VAR

// ---- Global Variables/InputsOutputs_CML/IOVariablesPACAN_CML.TcGVL
{attribute 'Tc2GvlVarNames'}
VAR_GLOBAL
(*TERMINAL 860KF1 - EL1008 ***********************************************************************)
	ib860KF1_1_FockeSignalPackAggregationTriggerCAM1			AT %I* : BOOL; (* 860KF1_1 *)
	ib860KF1_5_FockeSignalPackAggregationTriggerCAM2			AT %I* : BOOL; (* 860KF1_5 *)
	ib860KF1_2_FockeSignalPackAggregationTriggerCAM3			AT %I* : BOOL; (* 860KF1_2 *)
	ib860KF1_6_FockeSignalAutoRun								AT %I* : BOOL; (* 860KF1_6 *)
	ib860KF1_3_FockeSignalServoIndex 							AT %I* : BOOL; (* 860KF1_3 *)
	ib860KF1_7_FockeSignalMachineIndex 							AT %I* : BOOL; (* 860KF1_7 *)
	ib860KF1_4_FockeSignalPackRejected 							AT %I* : BOOL; (* 860KF1_4 *)
	ib860KF1_8_Spare 											AT %I* : BOOL; (* 860KF1_8 *)

(*TERMINAL 861KF1 - EL1008 ***********************************************************************)
	ib861KF1_1_FockeSignalStackerIndex							AT %I* : BOOL; (* 861KF1_1 *)
	ib861KF1_5_FockeSignalStackerIndex2							AT %I* : BOOL; (* 861KF1_5 *)
	ib861KF1_2_FockeSignalFilmIndex								AT %I* : BOOL; (* 861KF1_2 *)
	ib861KF1_6_FockeSignalMasterListTrigger						AT %I* : BOOL; (* 861KF1_6 *)
	ib861KF1_3_FockeSignalTriggerBackupCAM1_3					AT %I* : BOOL; (* 861KF1_3 *)
	ib861KF1_7_FockeSignalElevatorCameraTrigger					AT %I* : BOOL; (* 861KF1_7 *)
	ib861KF1_4_FockeSignalIntermediateCameraTrigger				AT %I* : BOOL; (* 861KF1_4 *)
	ib861KF1_8_FockeSignalTriggerBackupCAM1_3					AT %I* : BOOL; (* 861KF1_8 *)

(*TERMINAL 862KF1 - EL1008 ***********************************************************************)
	ib862KF1_1_FockeSignalPushIntoTurret						AT %I* : BOOL; (* 862KF1_1 *)
	ib862KF1_5_FockeSignalBuildBack								AT %I* : BOOL; (* 862KF1_5 *)
	ib862KF1_2_FockeSignalInfeedServoRunning					AT %I* : BOOL; (* 862KF1_2 *)
	ib862KF1_6_FockeSignalOuterAccepted							AT %I* : BOOL; (* 862KF1_6 *)
	ib660KF1_3_FockeSignalMachineRunning						AT %I* : BOOL; (* 862KF1_3 *)
	ib862KF1_7_FockeSignalFilmPresent							AT %I* : BOOL; (* 862KF1_7 *)
	ib862KF1_4_FockeSignalLightControlCamera					AT %I* : BOOL; (* 862KF1_4 *)
	ib862KF1_8_FockeSignalPrinterReady							AT %I* : BOOL; (* 862KF1_8 *)

(*TERMINAL 863KF1 - EL1008 ***********************************************************************)
	ib863KF1_1_FockeSignalRefeedServo							AT %I* : BOOL; (* 863KF1_1 *)
	ib863KF1_5_Spare											AT %I* : BOOL; (* 863KF1_5 *)
	ib863KF1_2_Spare											AT %I* : BOOL; (* 863KF1_2 *)
	ib863KF1_6_Spare											AT %I* : BOOL; (* 863KF1_6 *)
	ib863KF1_3_24VDCOK											AT %I* : BOOL; (* 863KF1_3 *)
	ib863KF1_7_Spare											AT %I* : BOOL; (* 863KF1_7 *)
	ib863KF1_4_Spare											AT %I* : BOOL; (* 863KF1_4 *)
	ib863KF1_8_Spare											AT %I* : BOOL; (* 863KF1_8 *)


(*TERMINAL 880KF1 - EL2008 ************************************************************************)
	qb880KF1_1_SignalToFockeReady								AT %Q* : BOOL; (* 880KF1_1 *)
	qb880KF1_5_SignalToFockeCutOut								AT %Q* : BOOL; (* 880KF1_5 *)
	qb880KF1_2_SignalToFockeRejectOuter							AT %Q* : BOOL; (* 880KF1_2 *)
	qb880KF1_6_SignalToFockeRejectLimitReachedTrigger			AT %Q* : BOOL; (* 880KF1_6 *)
	qb880KF1_3_SignalToFockeDynamicCameraTriggerPower			AT %Q* : BOOL; (* 880KF1_3 *)
	qb880KF1_7_Spare											AT %Q* : BOOL; (* 880KF1_7 *)
	qb880KF1_4_Spare											AT %Q* : BOOL; (* 880KF1_4 *)
	qb880KF1_8_Spare											AT %Q* : BOOL; (* 880KF1_8 *)

(*TERMINAL 881KF1 - EL2008 ************************************************************************)
	qb881KF1_1_MasterListCameraPower							AT %Q* : BOOL; (* 881KF1_1 *)
	qb881KF1_5_MasterListCameraTrigger							AT %Q* : BOOL; (* 881KF1_5 *)
	qb881KF1_2_AggregationCamera1Power							AT %Q* : BOOL; (* 881KF1_2 *)
	qb881KF1_6_AggregationCamera1Trigger						AT %Q* : BOOL; (* 881KF1_6 *)
	qb881KF1_3_AggregationCamera2Power							AT %Q* : BOOL; (* 881KF1_3 *)
	qb881KF1_7_AggregationCamera2Trigger						AT %Q* : BOOL; (* 881KF1_7 *)
	qb881KF1_4_AggregationCamera3Power							AT %Q* : BOOL; (* 881KF1_4 *)
	qb881KF1_8_AggregationCamera3Trigger						AT %Q* : BOOL; (* 881KF1_8 *)

(*TERMINAL 882KF1 - EL2008 ************************************************************************)
	qb882KF1_1_LightPoleGreen									AT %Q* : BOOL; (* 882KF1_1 *)
	qb882KF1_5_LightPoleAmber									AT %Q* : BOOL; (* 882KF1_5 *)
	qb882KF1_2_LightPoleRed										AT %Q* : BOOL; (* 882KF1_2 *)
	qb882KF1_6_LightPoleAlarm									AT %Q* : BOOL; (* 882KF1_6 *)
	qb882KF1_3_Spare											AT %Q* : BOOL; (* 882KF1_3 *)
	qb882KF1_7_Spare											AT %Q* : BOOL; (* 882KF1_7 *)
	qb882KF1_4_Spare											AT %Q* : BOOL; (* 882KF1_4 *)
	qb882KF1_8_Spare											AT %Q* : BOOL; (* 882KF1_8 *)
END_VAR

// ---- Global Variables/InputsOutputs_CML/IOVariablesPAOL_CML.TcGVL
{attribute 'Tc2GvlVarNames'}
VAR_GLOBAL

(*METS TPD - PAOL (CML) *)
(*TERMINAL 546KF1 - EK1100 ******************************************************)

(*TERMINAL 547KF2 - EL4002 ******************************************************)

	qn547KF1_1_LightingIntensity						AT %Q* : INT; (*547KF1_1*)
	qn547KF1_2_Spare								AT %Q* : INT; (*547KF1_2*)

(*TERMINAL 560KF1 - EL1008 ******************************************************)
	ib560KF1_1_PrePackAggregationCameraRigTrigger		AT %I* : BOOL; (* 560KF1_1 *)
	ib560KF1_5_PackAggregationCamera1Trigger			AT %I* : BOOL; (* 560KF1_5 *)
	ib560KF1_2_PackAggregationCamera2Trigger			AT %I* : BOOL; (* 560KF1_2 *)
	ib560KF1_6_PackAggregationCamera3Trigger			AT %I* : BOOL; (* 560KF1_6 *)
	ib560KF1_3_PreMachineBuildBack					AT %I* : BOOL; (* 560KF1_3 *)
	ib560KF1_7_TPDExitBlock							AT %I* : BOOL; (* 560KF1_7 *)
	ib560KF1_4_ConveyorIndexContact					AT %I* : BOOL; (* 560KF1_4 *)		(*not used on C922 and C925 *)
	ib560KF1_8_PackIsolatorDrive						AT %I* : BOOL; (* 560KF1_8 *)

(*TERMINAL 5480KF1 - EL2008 ******************************************************)
	qb580KF1_1_PackAggregationCamera1Enable			AT %Q* : BOOL; (* 580KF1_1 *)
	qb580KF1_5_PackAggregationCamera2Enable			AT %Q* : BOOL; (* 580KF1_5 *)
	qb580KF1_2_PackAggregationCamera3Enable			AT %Q* : BOOL; (* 580KF1_2 *)
	qb580KF1_6_PackAggregationCamera1Power			AT %Q* : BOOL; (* 580KF1_6 *)
	qb580KF1_3_PackAggregationCamera2Power			AT %Q* : BOOL; (* 580KF1_3 *)
	qb580KF1_7_PackAggregationCamera3Power			AT %Q* : BOOL; (* 580KF1_7 *)
	qb580KF1_4_Spare								AT %Q* : BOOL; (* 580KF1_4 *)
	qb580KF1_8_PackCamerasLenseAir					AT %Q* : BOOL; (* 580KF1_8 *)

END_VAR

// ---- Global Variables/InputsOutputs_CML/IOVariablesPLAS_CML.TcGVL
{attribute 'Tc2GvlVarNames'}
VAR_GLOBAL

(*TERMINAL XXXKF1 - EK1100 ******************************************************)


(*TERMINAL 747KF1 - EL4002 ******************************************************)
	qn747KF1_1_LightingIntensityPackAggregationCamera			AT %Q* : INT;
	qn747KF1_2_LightingIntensityPackConfirmationCamera			AT %Q* : INT;

(*TERMINAL 763KF1 - EL1008 ******************************************************)
	ib763KF1_1_MasterListCameraTrigSensor						AT %I* : BOOL;
	ib763KF1_5_SpareMasterListCameraTrigSensor					AT %I* : BOOL;		(* Option *)
	ib763KF1_2_AggregationCameraTrigSensor					AT %I* : BOOL;
	ib763KF1_6_SpareAggregationCamera1TrigSensor				AT %I* : BOOL;		(* Option *)
	ib763KF1_3_SpareAggregationCamera2TrigSensor				AT %I* : BOOL;		(* Option *)
	ib763KF1_7_PackQueueIndex								AT %I* : BOOL;
	ib763KF1_4_StackQueueIndex								AT %I* : BOOL; 		(* Option *)
	ib763KF1_8_SpareIndex									AT %I* : BOOL;		(* Option *)

(*TERMINAL 764KF1 - EL1008 ******************************************************)
	ib764KF1_1_OuterIndexComplete							AT %I* : BOOL;
	ib764KF1_5_SpareCameraTrigSensor							AT %I* : BOOL;		(* Option *)
	ib764KF1_2_Guard1 										AT %I* : BOOL;		(*FOCKE/GD Master list guard*)
	ib764KF1_6_Guard2										AT %I* : BOOL;		(*FOCKE/GD Master list guard*)
	ib764KF1_3_Guard3 										AT %I* : BOOL;		(*FOCKE/GD Aggregation guard*)
	ib764KF1_7_Guard4 										AT %I* : BOOL;		(*FOCKE/GD Aggregationt guard*) (*Option*)
	ib764KF1_4_OuterBrushOpen								AT %I* : BOOL;		(*Option*)
	ib764KF1_8_RejectTowerActive								AT %I* : BOOL;

(*TERMINAL 765KF1 (EL1008 8Ch. Dig. Input 24V, 3ms) ******************************************************)
	ib765KF1_1_FilmInPosition								AT %I*: BOOL;		(*Option*)
	ib765KF1_5_SparePrinterTrigger							AT %I*: BOOL;		(*Option*)
	ib765KF1_2_IntermediateCamera1TrigSesnor					AT %I*: BOOL;
	ib765KF1_6_HeatTunenelPackReject							AT %I*: BOOL;												(*not used on C922 and C925 *)
	ib765KF1_3_OuterAtAdditionalConveyor01 					AT %I*: BOOL;												(*not used on C922 and C925 *)
	ib765KF1_7_IntermediateCamera2TrigSesnor					AT %I*: BOOL;												(*not used on C922 and C925 *)
	ib765KF1_4_OuterAtReject								AT %I*: BOOL;		(*AdditionalConveyor01*)					(*not used on C922 and C925 *)
	ib765KF1_8_RejectConfirmation	 						AT %I*: BOOL;		(*AdditionalConveyor01*)					(*not used on C922 and C925 *)

(*TERMINAL 783KF1 - EL2008 ******************************************************)
	qb783KF1_1_MasterListCameraPower						AT %Q* : BOOL;
	qb783KF1_5_SpareMasterListCameraPower					AT %Q* : BOOL;		(* Option *)
	qb783KF1_2_SpareAggregationCameraPower					AT %Q* : BOOL;		(* Option *)
	qb783KF1_6_AggregationCamera1Power						AT %Q* : BOOL;
	qb783KF1_3_AggregationCamera2Power						AT %Q* : BOOL;
	qb783KF1_7_ConfirmationCamera1Power						AT %Q* : BOOL;
	qb783KF1_4_ConfirmationCamera2Power						AT %Q* : BOOL; 	(* Option *)
	qb783KF1_8_PLCControlledPackAggCamLightning			AT %Q* : BOOL;

(*TERMINAL 784KF1 - EL2008 ******************************************************)
	qb784KF1_1_MasterListCameraTrigger						AT %Q* : BOOL;
	qb784KF1_5_SpareMasterListCameraTrigger					AT %Q* : BOOL;		(* Option *)
	qb784KF1_2_AggregationCameraTrigger						AT %Q* : BOOL;
	qb784KF1_6_AggregationCamera1Trigger						AT %Q* : BOOL; 	(* Option *)
	qb784KF1_3_AggregationCamera2Trigger						AT %Q* : BOOL; 	(* Option *)
	qb784KF1_7_ConfirmationCamera1Trigger					AT %Q* : BOOL;
	qb784KF1_4_ConfirmationCamera2Trigger					AT %Q* : BOOL; 	(* Option *)
	qb784KF1_8_PLCControlledPackConfirmCamLightning		AT %Q* : BOOL;

(*TERMINAL 785KF1 (EL2008 8Ch. Dig. Output 24V, 3ms) ******************************************************)
	qb785KF1_1_IntermediateCamera1Trigger					AT %Q*: BOOL;
	qb785KF1_5_IntermediateCamera1Power					AT %Q*: BOOL;
	qb785KF1_2_IntermediateCamera2Trigger					AT %Q*: BOOL;												(*not used on C922 and C925 *)
	qb785KF1_6_IntermediateCamera3Power					AT %Q*: BOOL;												(*not used on C922 and C925 *)
	qb785KF1_3_RejectCylinderExtended						AT %Q*: BOOL;			(*AdditionalConveyor01*)				(*not used on C922 and C925 *)
	qb785KF1_7_RjectCylinderRetracted							AT %Q*: BOOL;			(*AdditionalConveyor01*)				(*not used on C922 and C925 *)
	qb785KF1_4_IntermediateCamera3Trigger					AT %Q*: BOOL;												(*not used on C922 and C925 *)
	qb785KF1_8_IntermediateCamera3Power					AT %Q*: BOOL;												(*not used on C922 and C925 *)

END_VAR

// ---- Global Variables/InputsOutputs_OC/IOVariablesCX_OC.TcGVL
{attribute 'Tc2GvlVarNames'}
VAR_GLOBAL
(***************************Terminal States Diagnostic*****************************************************)

	istEtherCATMasterState							AT	%I*	: ST_CX_EtherCATMasterState;
	iaEtherCATSlaveState							AT 	%I*	: ARRAY [0..cMAX_ETHERCAT_SLAVES] OF UINT;

(*****************************Input/Output Cards*********************************************************)

	(*TERMINAL 45KF2 (EK1200-5000 EtherCAT Power supply (2A E-Bus)) ***************************************)

